TYPE _eDbmText : (txt_DbVar_C0_RamEcuInputsC0_PressureBlockOscillationState_0 := 0, txt_DbVar_C0_RamEcuInputsC0_PressureBlockOscillationValue_0 := 1, txt_DbVar_C0_RamEcuInputsC0_PressureBlockOscillationRawValue_0 := 2, txt_DbVar_C0_RamEcuInputsC0_PressureBrakeSensorState_0 := 3, txt_DbVar_C0_RamEcuInputsC0_PressureBrakeSensorValue_0 := 4, txt_DbVar_C0_RamEcuInputsC0_PressureBrakeSensorRawValue_0 := 5, txt_DbVar_C0_RamEcuInputsC0_TemperatureTransmissionState_0 := 6, txt_DbVar_C0_RamEcuInputsC0_TemperatureTransmissionValue_0 := 7, txt_DbVar_C0_RamEcuInputsC0_TemperatureTransmissionRawValue_0 := 8, txt_DbVar_C0_RamEcuInputsC0_FaultPvgLeftTrakState_0 := 9, txt_DbVar_C0_RamEcuInputsC0_FaultPvgLeftTrakRawValue_0 := 10, txt_DbVar_C0_RamEcuInputsC0_FaultPvgRightTrakState_0 := 11, txt_DbVar_C0_RamEcuInputsC0_FaultPvgRightTrakRawValue_0 := 12, txt_DbVar_C0_RamEcuInputsC0_DownAxleOscillantState_0 := 13, txt_DbVar_C0_RamEcuInputsC0_DownAxleOscillantRawValuePin0_0 := 14, txt_DbVar_C0_RamEcuInputsC0_DownAxleOscillantRawValuePin1_0 := 15, txt_DbVar_C0_RamEcuInputsC0_DownAxleFixeState_0 := 16, txt_DbVar_C0_RamEcuInputsC0_DownAxleFixeRawValuePin0_0 := 17, txt_DbVar_C0_RamEcuInputsC0_DownAxleFixeRawValuePin1_0 := 18, txt_DbVar_C0_RamEcuInputsC0_UpAxleOscillantState_0 := 19, txt_DbVar_C0_RamEcuInputsC0_UpAxleOscillantRawValue_0 := 20, txt_DbVar_C0_RamEcuInputsC0_UpAxleFixeState_0 := 21, txt_DbVar_C0_RamEcuInputsC0_UpAxleFixeRawValue_0 := 22, txt_DbVar_C0_RamEcuInputsC0_FrameRotationSensor1State_0 := 23, txt_DbVar_C0_RamEcuInputsC0_FrameRotationSensor1RawValuePin0_0 := 24, txt_DbVar_C0_RamEcuInputsC0_FrameRotationSensor1RawValuePin1_0 := 25, txt_DbVar_C0_RamEcuInputsC0_RailHookSensorState_0 := 26, txt_DbVar_C0_RamEcuInputsC0_RailHookSensorRawValue_0 := 27, txt_DbVar_C0_RamEcuInputsC0_InductiveRailSensorState_0 := 28, txt_DbVar_C0_RamEcuInputsC0_InductiveRailSensorRawValue_0 := 29, txt_DbVar_C0_RamEcuInputsC0_CenteredTurretState_0 := 30, txt_DbVar_C0_RamEcuInputsC0_CenteredTurretRawValue_0 := 31, txt_DbVar_C0_RamEcuInputsC0_WorkKeyTrackSideState_0 := 32, txt_DbVar_C0_RamEcuInputsC0_WorkKeyTrackSideRawValue_0 := 33, txt_DbVar_C0_RamEcuInputsC0_FrameRotationSensor2State_0 := 34, txt_DbVar_C0_RamEcuInputsC0_FrameRotationSensor2RawValuePin0_0 := 35, txt_DbVar_C0_RamEcuInputsC0_FrameRotationSensor2RawValuePin1_0 := 36, txt_DbVar_C0_RamEcuInputsC0_WorkKeyBilateralState_0 := 37, txt_DbVar_C0_RamEcuInputsC0_WorkKeyBilateralRawValue_0 := 38, txt_DbVar_C0_RamEcuInputsC0_WorkKeyCentredState_0 := 39, txt_DbVar_C0_RamEcuInputsC0_WorkKeyCentredRawValue_0 := 40, txt_DbVar_C0_RamEcuInputsC0_AbutmentTurretTrackSideState_0 := 41, txt_DbVar_C0_RamEcuInputsC0_AbutmentTurretTrackSideRaw_0 := 42, txt_DbVar_C0_RamEcuInputsC0_AbutmentTurretCentredSideState_0 := 43, txt_DbVar_C0_RamEcuInputsC0_AbutmentTurretCentredSideRaw_0 := 44, txt_DbVar_C0_RamEcuInputsC0_OscillantAxleSpeedSensorDirState_0 := 45, txt_DbVar_C0_RamEcuInputsC0_OscillantAxleSpeedSensorDirRaw_0 := 46, txt_DbVar_C0_RamEcuInputsC0_FixeAxleSpeedSensorDirState_0 := 47, txt_DbVar_C0_RamEcuInputsC0_FixeAxleSpeedSensorDirRaw_0 := 48, txt_DbVar_C0_RamEcuInputsC0_TrailerGacheState_0 := 49, txt_DbVar_C0_RamEcuInputsC0_TrailerGacheRawValue_0 := 50, txt_DbVar_C0_RamEcuInputsC0_MeasuringMastSensorFoldedState_0 := 51, txt_DbVar_C0_RamEcuInputsC0_MeasuringMastSensorFoldedRaw_0 := 52, txt_DbVar_C0_RamEcuInputsC0_OscillantAxleFrequency_0 := 53, txt_DbVar_C0_RamEcuInputsC0_FixeAxleFrequency_0 := 54, txt_DbVar_C0_RamEcuInputsC0_AruRadio1ContactState_0 := 55, txt_DbVar_C0_RamEcuInputsC0_AruRadio1ContactRawValue_0 := 56, txt_DbVar_C0_RamEcuInputsC0_AruRadio2ContactState_0 := 57, txt_DbVar_C0_RamEcuInputsC0_AruRadio2ContactRawValue_0 := 58, txt_DbVar_C0_RamEcuInputsC0_Aru1ContactState_0 := 59, txt_DbVar_C0_RamEcuInputsC0_Aru1ContactRawValue_0 := 60, txt_DbVar_C0_RamEcuInputsC0_Aru2ContactState_0 := 61, txt_DbVar_C0_RamEcuInputsC0_Aru2ContactRawValue_0 := 62, txt_DbVar_C0_RamEcuInputsC0_StarterMotorState_0 := 63, txt_DbVar_C0_RamEcuInputsC0_StarterMotorRawValue_0 := 64, txt_DbVar_C0_RamEcuInputsC0_AutorisationHighSpeedKeyState_0 := 65, txt_DbVar_C0_RamEcuInputsC0_AutorisationHighSpeedKeyRawValue_0 := 66, txt_DbVar_C0_RamEcuInputsC0_ElectricPumpPressureState_0 := 67, txt_DbVar_C0_RamEcuInputsC0_ElectricPumpPressureValue_0 := 68, txt_DbVar_C0_RamEcuInputsC0_ElectricPumpPressureRawValue_0 := 69, txt_DbVar_C0_RamEcuInputsC0_UpMastSensorNCState_0 := 70, txt_DbVar_C0_RamEcuInputsC0_UpMastSensorNCRawValue_0 := 71, txt_DbVar_C0_RamEcuInputsC0_ValveInDownPositionSensorState_0 := 72, txt_DbVar_C0_RamEcuInputsC0_ValveInDownPositionSensorValue_0 := 73, txt_DbVar_C0_RamEcuOutputsC0_EvDeflectorTransmissionCommand_0 := 74, txt_DbVar_C0_RamEcuOutputsC0_EvDeflectorTransmissionValue_0 := 75, txt_DbVar_C0_RamEcuOutputsC0_EvUpMeasuringMastCommand_0 := 76, txt_DbVar_C0_RamEcuOutputsC0_EvUpMeasuringMastValue_0 := 77, txt_DbVar_C0_RamEcuOutputsC0_EvDownMeasuringMastCommand_0 := 78, txt_DbVar_C0_RamEcuOutputsC0_EvDownMeasuringMastValue_0 := 79, txt_DbVar_C0_RamEcuOutputsC0_EvServiceBrakeTrackCommand_0 := 80, txt_DbVar_C0_RamEcuOutputsC0_EvServiceBrakeTrackValue_0 := 81, txt_DbVar_C0_RamEcuOutputsC0_EvPowerReductionCommand_0 := 82, txt_DbVar_C0_RamEcuOutputsC0_EvPowerReductionValue_0 := 83, txt_DbVar_C0_RamEcuOutputsC0_EvFrameRotation1Command_0 := 84, txt_DbVar_C0_RamEcuOutputsC0_EvFrameRotation1Value_0 := 85, txt_DbVar_C0_RamEcuOutputsC0_EvFrameRotation2Command_0 := 86, txt_DbVar_C0_RamEcuOutputsC0_EvFrameRotation2Value_0 := 87, txt_DbVar_C0_RamEcuOutputsC0_SupplyRadioReceiverCommand_0 := 88, txt_DbVar_C0_RamEcuOutputsC0_SupplyRadioReceiverValue_0 := 89, txt_DbVar_C0_RamEcuOutputsC0_BuzzerLynxMovingMachineCommand_0 := 90, txt_DbVar_C0_RamEcuOutputsC0_BuzzerLynxMovingMachineValue_0 := 91, txt_DbVar_C0_RamEcuOutputsC0_WhiteLightsTrailerCommand_0 := 92, txt_DbVar_C0_RamEcuOutputsC0_WhiteLightsTrailerValue_0 := 93, txt_DbVar_C0_RamEcuOutputsC0_RedLightsTrailerCommand_0 := 94, txt_DbVar_C0_RamEcuOutputsC0_RedLightsTrailerValue_0 := 95, txt_DbVar_C0_RamEcuOutputsC0_WhiteLightAVGCommand_0 := 96, txt_DbVar_C0_RamEcuOutputsC0_WhiteLightAVGValue_0 := 97, txt_DbVar_C0_RamEcuOutputsC0_WhiteLightAVDCommand_0 := 98, txt_DbVar_C0_RamEcuOutputsC0_WhiteLightAVDValue_0 := 99, txt_DbVar_C0_RamEcuOutputsC0_RedLightAVGCommand_0 := 100, txt_DbVar_C0_RamEcuOutputsC0_RedLightAVGValue_0 := 101, txt_DbVar_C0_RamEcuOutputsC0_RedLightAVDCommand_0 := 102, txt_DbVar_C0_RamEcuOutputsC0_RedLightAVDValue_0 := 103, txt_DbVar_C0_RamEcuOutputsC0_WhiteLightARGCommand_0 := 104, txt_DbVar_C0_RamEcuOutputsC0_WhiteLightARGValue_0 := 105, txt_DbVar_C0_RamEcuOutputsC0_WhiteLightARDCommand_0 := 106, txt_DbVar_C0_RamEcuOutputsC0_WhiteLightARDValue_0 := 107, txt_DbVar_C0_RamEcuOutputsC0_RedLightARGCommand_0 := 108, txt_DbVar_C0_RamEcuOutputsC0_RedLightARGValue_0 := 109, txt_DbVar_C0_RamEcuOutputsC0_RedLightARDCommand_0 := 110, txt_DbVar_C0_RamEcuOutputsC0_RedLightARDValue_0 := 111, txt_DbVar_C0_RamEcuOutputsC0_SupllyPvgLeftTrackCommand_0 := 112, txt_DbVar_C0_RamEcuOutputsC0_SupllyPvgLeftTrackValue_0 := 113, txt_DbVar_C0_RamEcuOutputsC0_SupllyPvgRightTrackCommand_0 := 114, txt_DbVar_C0_RamEcuOutputsC0_SupllyPvgRightTrackValue_0 := 115, txt_DbVar_C0_RamEcuOutputsC0_EvUnBlockOscillationAxleState_0 := 116, txt_DbVar_C0_RamEcuOutputsC0_EvUnBlockOscillationAxleCmdBool_0 := 117, txt_DbVar_C0_RamEcuOutputsC0_EvUpAxleOscillantState_0 := 118, txt_DbVar_C0_RamEcuOutputsC0_EvUpAxleOscillantCommandBool_0 := 119, txt_DbVar_C0_RamEcuOutputsC0_EvDownAxleOscillantState_0 := 120, txt_DbVar_C0_RamEcuOutputsC0_EvDownAxleOscillantCommandBool_0 := 121, txt_DbVar_C0_RamEcuOutputsC0_EvUpAxleFixeState_0 := 122, txt_DbVar_C0_RamEcuOutputsC0_EvUpAxleFixeCommandBool_0 := 123, txt_DbVar_C0_RamEcuOutputsC0_EvDownAxleFixeState_0 := 124, txt_DbVar_C0_RamEcuOutputsC0_EvDownAxleFixeCommandBool_0 := 125, txt_DbVar_C0_RamEcuOutputsC0_EvParkBrakeAxleOscillantState_0 := 126, txt_DbVar_C0_RamEcuOutputsC0_EvParkBrakeAxleOscillantCmdBool_0 := 127, txt_DbVar_C0_RamEcuOutputsC0_EvParkBrakeAxleFixeState_0 := 128, txt_DbVar_C0_RamEcuOutputsC0_EvParkBrakeAxleFixeCmdBool_0 := 129, txt_DbVar_C0_RamEcuOutputsC0_EvServiceBrakeAxleOscillantState_0 := 130, txt_DbVar_C0_RamEcuOutputsC0_EvServiceBrakeAxleOsciCmdBool_0 := 131, txt_DbVar_C0_RamEcuOutputsC0_EvServiceBrakeAxleFixeState_0 := 132, txt_DbVar_C0_RamEcuOutputsC0_EvServiceBrakeAxleFixeCmdBool_0 := 133, txt_DbVar_C0_RamEcuOutputsC0_KlaxonNeotecState_0 := 134, txt_DbVar_C0_RamEcuOutputsC0_KlaxonNeotecCmdBool_0 := 135, txt_DbVar_C0_RamEcuOutputsC0_ForwardPumpState_0 := 136, txt_DbVar_C0_RamEcuOutputsC0_ForwardPumpCommand_0 := 137, txt_DbVar_C0_RamEcuOutputsC0_ForwardPumpCurrent_0 := 138, txt_DbVar_C0_RamEcuOutputsC0_BackwardPumpState_0 := 139, txt_DbVar_C0_RamEcuOutputsC0_BackwardPumpCommand_0 := 140, txt_DbVar_C0_RamEcuOutputsC0_BackwardPumpCurrent_0 := 141, txt_DbVar_C0_RamEcuOutputsC0_PvgLeftTrackCommand_0 := 142, txt_DbVar_C0_RamEcuOutputsC0_PvgLeftTrackVoltage_0 := 143, txt_DbVar_C0_RamEcuOutputsC0_PvgRightTrackCommand_0 := 144, txt_DbVar_C0_RamEcuOutputsC0_PvgRightTrackVoltage_0 := 145, txt_DbVar_C0_RamEcuOutputsC0_SupplyAnaSensorsCommand_0 := 146, txt_DbVar_C0_RamEcuOutputsC0_SupplyAnaSensorsValue_0 := 147, txt_DbVar_C0_RamEcuOutputsC0_PvgLeftTrackLowsideCommand_0 := 148, txt_DbVar_C0_RamEcuOutputsC0_PvgLeftTrackLowsideValue_0 := 149, txt_DbVar_C0_RamEcuOutputsC0_PvgRightTrackLowsideCommand_0 := 150, txt_DbVar_C0_RamEcuOutputsC0_PvgRightTrackLowsideValue_0 := 151, txt_DbVar_C0_RamEcuOutputsC0_ReturnLowSideEvForwardPumpCmd_0 := 152, txt_DbVar_C0_RamEcuOutputsC0_ReturnLowSideEvForwardPumpState_0 := 153, txt_DbVar_C0_RamEcuOutputsC0_ReturnLowSideEvBackwardPumpCmd_0 := 154, txt_DbVar_C0_RamEcuOutputsC0_ReturnLowSideEvBackwardPumpState_0 := 155, txt_DbVar_C0_RamEcuOutputsC0_NeonLightsCmd_0 := 156, txt_DbVar_C0_RamEcuOutputsC0_NeonLightsValue_0 := 157, txt_DbVar_C0_RamEcuOutputsC0_Ev2DeflectorTransmissionValue_0 := 158, txt_DbVar_C0_RamEcuOutputsC0_CoolingRelayCommand_0 := 159, txt_DbVar_C0_RamEcuOutputsC0_CoolingRelayState_0 := 160, txt_DbVar_C0_RamEcuOutputsC0_Ev2ndParkBrakeAxleFixe_0 := 161, txt_DbVar_C0_RamEcuOutputsC0_Ev2ndParkBrakeAxleOsci_0 := 162, txt_DbVar_C0_RamEcuOutputsC0_Ev2ndParkBrakeAxleFixeState_0 := 163, txt_DbVar_C0_RamEcuOutputsC0_Ev2ndParkBrakeAxleOsciState_0 := 164, txt_DbVar_C0_RamEcuOutputsC0_PvgTransRailElectricCmd_0 := 165, txt_DbVar_C0_RamEcuOutputsC0_PvgTransRailElectricVoltage_0 := 166, txt_DbVar_C0_RamEcuOutputsC0_SupllyPvgTransRailElectricCmd_0 := 167, txt_DbVar_C0_RamEcuOutputsC0_SupllyPvgTransRailElectricState_0 := 168, txt_DbVar_C0_RamEcuOutputsC0_EvDevRailElectricModeCmd_0 := 169, txt_DbVar_C0_RamEcuOutputsC0_EvDevRailElectricModeState_0 := 170, txt_DbVar_C0_RamEcuOutputsC0_RelayCutOffVariatorElectricCmd_0 := 171, txt_DbVar_C0_RamEcuOutputsC0_RelayCutOffVariatorElectricState_0 := 172, txt_DbVar_C0_RamEcuOutputsC0_RelayEnableBatteryCmd_0 := 173, txt_DbVar_C0_RamEcuOutputsC0_RelayEnableBatteryState_0 := 174, txt_DbVar_C0_RamGeneralC0_LifeByte_0 := 175, txt_DbVar_C0_RamGeneralC0_WatchdogState_0 := 176, txt_DbVar_C0_RamGeneralC0_EcuVoltage_0 := 177, txt_DbVar_C0_RamGeneralC0_OffRailMode_0 := 178, txt_DbVar_C0_RamGeneralC0_RailSpeedMode_0 := 179, txt_DbVar_C0_RamGeneralC0_OutputLutLeftManipulator_0 := 180, txt_DbVar_C0_RamGeneralC0_OutputLutLeftTrackPvg_0 := 181, txt_DbVar_C0_RamGeneralC0_OutputLutRightManipulator_0 := 182, txt_DbVar_C0_RamGeneralC0_OutputLutRightTrackPvg_0 := 183, txt_DbVar_C0_RamGeneralC0_OutputLutJoystickAdvanceRail_0 := 184, txt_DbVar_C0_RamGeneralC0_OutputLutForwardPumpTransmission_0 := 185, txt_DbVar_C0_RamGeneralC0_OutputLutBackwardPumpTransm_0 := 186, txt_DbVar_C0_RamGeneralC0_ConsigneForwardPumpTransmPercent_0 := 187, txt_DbVar_C0_RamGeneralC0_LastJoystickAdvanceValue_0 := 188, txt_DbVar_C0_RamGeneralC0_JoystickAdvanceScalingValue_0 := 189, txt_DbVar_C0_RamGeneralC0_StateServiceBrakeRail_0 := 190, txt_DbVar_C0_RamGeneralC0_EnableStartTimerServiceBrake_0 := 191, txt_DbVar_C0_RamGeneralC0_SpeedMotorCommandTest_0 := 192, txt_DbVar_C0_RamGeneralC0_ForceSilentModeMotorTest_0 := 193, txt_DbVar_C0_RamGeneralC0_AngularSensorTest_0 := 194, txt_DbVar_C0_RamGeneralC0_SpeedAxleSensor_0 := 195, txt_DbVar_C0_RamGeneralC0_AverageTimeCycle_0 := 196, txt_DbVar_C0_RamGeneralC0_MaxTimeCycle_0 := 197, txt_DbVar_C0_RamGeneralC0_FirstTranslationReleaseParkBrake_0 := 198, txt_DbVar_C0_RamGeneralC0_AutorizeUpAxleOscillant_0 := 199, txt_DbVar_C0_RamGeneralC0_AutorizeDownAxleOscillant_0 := 200, txt_DbVar_C0_RamGeneralC0_AutorizeUpAxlefixe_0 := 201, txt_DbVar_C0_RamGeneralC0_AutorizeDownAxlefixe_0 := 202, txt_DbVar_C0_RamGeneralC0_EngineOn_0 := 203, txt_DbVar_C0_RamGeneralC0_TranslationMovementIsSolicited_0 := 204, txt_DbVar_C0_RamGeneralC0_RailTranslationDirection_0 := 205, txt_DbVar_C0_RamGeneralC0_SetConditionAruRadioAlarm_0 := 206, txt_DbVar_C0_RamGeneralC0_JoystickAdvanceSetpointAfterRamp_0 := 207, txt_DbVar_C0_RamGeneralC0_StabilizedStop_0 := 208, txt_DbVar_C0_RamGeneralC0_EmergencyBrake_0 := 209, txt_DbVar_C0_RamGeneralC0_EmergencyServiceBrakeTimerDone_0 := 210, txt_DbVar_C0_RamGeneralC0_StoppedMachineUnblkOsciTimerDone_0 := 211, txt_DbVar_C0_RamGeneralC0_OutLutLeftManipulatorAfterRamp_0 := 212, txt_DbVar_C0_RamGeneralC0_OutLutRightManipulatorAfterRamp_0 := 213, txt_DbVar_C0_RamGeneralC0_DeltaBeetweenLeftRightPvgCrawler_0 := 214, txt_DbVar_C0_RamGeneralC0_ConsigneLeftPvgTrack_0 := 215, txt_DbVar_C0_RamGeneralC0_ConsigneRightPvgTrack_0 := 216, txt_DbVar_C0_RamGeneralC0_BrakeWithoutGachetteOrPedal_0 := 217, txt_DbVar_C0_RamGeneralC0_AruRadioAlarmCounter_0 := 218, txt_DbVar_C0_RamGeneralC0_RedLightARGBasketCmd_0 := 219, txt_DbVar_C0_RamGeneralC0_WhiteLightARGBasketCmd_0 := 220, txt_DbVar_C0_RamGeneralC0_PortillonLadderClose_0 := 221, txt_DbVar_C0_RamGeneralC0_TestEvision_0 := 222, txt_DbVar_C0_RamGeneralC0_PosJoystickAdvance_0 := 223, txt_DbVar_C0_RamGeneralC0_RetainPosJoyAdvanceUntilBrake_0 := 224, txt_DbVar_C0_RamGeneralC0_AuthorizeForwardCrawler_0 := 225, txt_DbVar_C0_RamGeneralC0_AuthorizeBackwardCrawler_0 := 226, txt_DbVar_C0_RamGeneralC0_ReturnValueUartInit_0 := 227, txt_DbVar_C0_RamGeneralC0_AuthorizeTransRailMovement_0 := 228, txt_DbVar_C0_RamGeneralC0_EvForwardTrackConsigne_0 := 229, txt_DbVar_C0_RamGeneralC0_EvForwardRailConsigne_0 := 230, txt_DbVar_C0_RamGeneralC0_EngineTimeSecond_0 := 231, txt_DbVar_C0_RamGeneralC0_RamGeneralNeotecC0_1_0 := 232, txt_DbVar_C0_RamGeneralC0_RamGeneralNeotecC0_1_1_0 := 233, txt_DbVar_C0_RamGeneralC0_RamGeneralNeotecC0_1_2_0 := 234, txt_DbVar_C0_RamGeneralC0_RamGeneralNeotecC0_1_3_0 := 235, txt_DbVar_C0_RamGeneralC0_RamGeneralNeotecC0_1_4_0 := 236, txt_DbVar_C0_RamGeneralC0_RamGeneralNeotecC0_1_5_0 := 237, txt_DbVar_C0_RamGeneralC0_RamGeneralNeotecC0_1_6_0 := 238, txt_DbVar_C0_RamGeneralC0_RamGeneralNeotecC0_1_7_0 := 239, txt_DbVar_C0_RamGeneralC0_RamGeneralNeotecC0_1_8_0 := 240, txt_DbVar_C0_RamGeneralC0_RamGeneralNeotecC0_1_9_0 := 241, txt_DbVar_C0_RamGeneralC0_RamGeneralNeotecC0_1_10_0 := 242, txt_DbVar_C0_RamGeneralC0_RamGeneralNeotecC0_1_11_0 := 243, txt_DbVar_C0_RamGeneralC0_RamGeneralNeotecC0_1_12_0 := 244, txt_DbVar_C0_RamGeneralC0_RamGeneralNeotecC0_1_13_0 := 245, txt_DbVar_C0_RamGeneralC0_RamGeneralNeotecC0_1_14_0 := 246, txt_DbVar_C0_RamGeneralC0_RamGeneralNeotecC0_1_15_0 := 247, txt_DbVar_C0_RamGeneralC0_RamGeneralNeotecC0_2_0 := 248, txt_DbVar_C0_RamGeneralC0_RamGeneralNeotecC0_2_1_0 := 249, txt_DbVar_C0_RamGeneralC0_RamGeneralNeotecC0_2_2_0 := 250, txt_DbVar_C0_RamGeneralC0_RamGeneralNeotecC0_2_3_0 := 251, txt_DbVar_C0_RamGeneralC0_RamGeneralNeotecC0_2_4_0 := 252, txt_DbVar_C0_RamGeneralC0_RamGeneralNeotecC0_2_5_0 := 253, txt_DbVar_C0_RamGeneralC0_RamGeneralNeotecC0_3_0 := 254, txt_DbVar_C0_RamGeneralC0_RamGeneralNeotecC0_3_1_0 := 255, txt_DbVar_C0_RamGeneralC0_RamGeneralNeotecC0_3_2_0 := 256, txt_DbVar_C0_RamGeneralC0_RamGeneralNeotecC0_3_3_0 := 257, txt_DbVar_C0_RamGeneralC0_RamGeneralNeotecC0_3_4_0 := 258, txt_DbVar_C0_RamGeneralC0_RamGeneralNeotecC0_3_5_0 := 259, txt_DbVar_C0_RamGeneralC0_RamGeneralNeotecC0_3_6_0 := 260, txt_DbVar_C0_RamGeneralC0_RamGeneralNeotecC0_3_7_0 := 261, txt_DbVar_C0_RamGeneralC0_RamGeneralNeotecC0_3_8_0 := 262, txt_DbVar_C0_RamGeneralC0_RamGeneralNeotecC0_4_0 := 263, txt_DbVar_C0_RamGeneralC0_RamGeneralNeotecC0_4_1_0 := 264, txt_DbVar_C0_RamGeneralC0_RamGeneralNeotecC0_4_2_0 := 265, txt_DbVar_C0_RamGeneralC0_RamGeneralNeotecC0_4_3_0 := 266, txt_DbVar_C0_RamGeneralC0_RamGeneralNeotecC0_4_4_0 := 267, txt_DbVar_C0_RamGeneralC0_RamGeneralNeotecC0_4_5_0 := 268, txt_DbVar_C0_RamGeneralC0_RamGeneralNeotecC0_4_6_0 := 269, txt_DbVar_C0_RamGeneralC0_RamGeneralNeotecC0_4_7_0 := 270, txt_DbVar_C0_RamGeneralC0_RamGeneralNeotecC0_4_8_0 := 271, txt_DbVar_C0_RamGeneralC0_RedLightARDBasketCmd_0 := 272, txt_DbVar_C0_RamGeneralC0_WhiteLightARDBasketCmd_0 := 273, txt_DbVar_C0_RamGeneralC0_ActiveFailure_0 := 274, txt_DbVar_C0_RamGeneralC0_ReductionPumpRail_0 := 275, txt_DbVar_C0_RamGeneralC0_ReductionPumpTrack_0 := 276, txt_DbVar_C0_RamGeneralC0_ActiveWhiteLights15746_0 := 277, txt_DbVar_C0_RamGeneralC0_WhiteLightAv15746Command_0 := 278, txt_DbVar_C0_RamGeneralC0_WhiteLightAr15746Command_0 := 279, txt_DbVar_C0_RamGeneralC0_TestElectricalIO_0 := 280, txt_DbVar_C0_RamGeneralC0_SendEventDataloggerMessage_0 := 281, txt_DbVar_C0_RamGeneralC0_SlopeModeFromC1_0 := 282, txt_DbVar_C0_RamGeneralC0_BlinkLow_0 := 283, txt_DbVar_C0_RamGeneralC0_TotalDistance_0 := 284, txt_DbVar_C0_RamGeneralC0_RunningStable48XS_0 := 285, txt_DbVar_C0_RamGeneralC0_AlarmHydTempRailActive_0 := 286, txt_DbVar_C0_RamGeneralC0_AlarmHydTempCrawlerActive_0 := 287, txt_DbVar_C0_RamGeneralC0_FaultyValue_0 := 288, txt_DbVar_C0_RamGeneralC0_DeviceNum_0 := 289, txt_DbVar_C0_RamGeneralC0_ErrorCode_0 := 290, txt_DbVar_C0_RamGeneralC0_EngineRunningStable_0 := 291, txt_DbVar_C0_NvOptionsC0_ConfigHollandaise_0 := 292, txt_DbVar_C0_NvOptionsC0_Portillon_0 := 293, txt_DbVar_C0_NvOptionsC0_Ladder_0 := 294, txt_DbVar_C0_NvOptionsC0_MeasuringMat_0 := 295, txt_DbVar_C0_NvOptionsC0_IncliBasketHighSectorForAcesSite_0 := 296, txt_DbVar_C0_NvOptionsC0_BasketCenteredForAccesSite_0 := 297, txt_DbVar_C0_NvOptionsC0_MastDigitalDisplay_0 := 298, txt_DbVar_C0_NvOptionsC0_AutorisationWorkKeyPresent_0 := 299, txt_DbVar_C0_NvOptionsC0_SecondParkBrakeActive_0 := 300, txt_DbVar_C0_NvOptionsC0_AddPerformanceFunc_0 := 301, txt_DbVar_C0_NvOptionsC0_BasketTurretLimitation_0 := 302, txt_DbVar_C0_NvOptionsC0_PresenceSensorPlate_0 := 303, txt_DbVar_C0_NvMemoryC0_NCycleBrakePerform_0 := 304, txt_DbVar_C0_NvMemoryC0_LightMode_0 := 305, txt_DbVar_C0_NvMemoryC0_VarMemory1_0 := 306, txt_DbVar_C0_NvMemoryC0_VarMemory2_0 := 307, txt_DbVar_C0_NvMemoryC0_VarMemory3_0 := 308, txt_DbVar_C0_NvMemoryC0_VarMemory4_0 := 309, txt_DbVar_C0_NvMemoryC0_VarMemory5_0 := 310, txt_DbVar_C0_NvMemoryC0_VarMemory6_0 := 311, txt_DbVar_C0_NvMemoryC0_VarMemory7_0 := 312, txt_DbVar_C0_NvMemoryC0_VarMemory8_0 := 313, txt_DbVar_C0_NvMemoryC0_VarMemory9_0 := 314, txt_DbVar_C0_NvMemoryC0_VarMemory10_0 := 315, txt_DbVar_C0_NvMemoryC0_VarMemory11_0 := 316, txt_DbVar_C0_NvMemoryC0_VarMemory12_0 := 317, txt_DbVar_C0_NvMemoryC0_VarMemory13_0 := 318, txt_DbVar_C0_NvMemoryC0_VarMemory14_0 := 319, txt_DbVar_C0_NvMemoryC0_gDistanceTraveledMeasureMast_0 := 320, txt_DbVar_C0_NvMemoryC0_NCycle2ndParkBrakePerform_0 := 321, txt_DbVar_C0_NvMemoryC0_gTotalDistanceMsb_0 := 322, txt_DbVar_C0_NvMemoryC0_gTotalDistanceLsb_0 := 323, txt_DbVar_C0_NvParametersC0_LimitTresholdAngleRadioControl_0 := 324, txt_DbVar_C0_NvParametersC0_TresholdMinimalSpeedParkBrake_0 := 325, txt_DbVar_C0_NvParametersC0_TresholdMinimalSpeedServiceBrake_0 := 326, txt_DbVar_C0_NvParametersC0_AdditionnalPourcentFwardPumpCmd_0 := 327, txt_DbVar_C0_NvParametersC0_AddPrctFwardPumpSilentModeMotor_0 := 328, txt_DbVar_C0_NvParametersC0_NodeIdRadioCommand_0 := 329, txt_DbVar_C0_NvParametersC0_DeadZoneJoystickRotationTurret_0 := 330, txt_DbVar_C0_NvParametersC0_ServiceAxleBrakeTimeBeforeBrake_0 := 331, txt_DbVar_C0_NvParametersC0_ServiceBrakeOffrailTime_0 := 332, txt_DbVar_C0_NvParametersC0_EngineOffCurEvForwardPump_0 := 333, txt_DbVar_C0_NvParametersC0_MinCurEvForwardPump_0 := 334, txt_DbVar_C0_NvParametersC0_StopCurEvForwardPump_0 := 335, txt_DbVar_C0_NvParametersC0_EngineOffCurEvBackwardPump_0 := 336, txt_DbVar_C0_NvParametersC0_MinCurEvBackwardPump_0 := 337, txt_DbVar_C0_NvParametersC0_StopCurEvBackwardPump_0 := 338, txt_DbVar_C0_NvParametersC0_PosNeutralJoyAdvancement_0 := 339, txt_DbVar_C0_NvParametersC0_PidGpEvForwardPump_0 := 340, txt_DbVar_C0_NvParametersC0_PidTiEvForwardPump_0 := 341, txt_DbVar_C0_NvParametersC0_PidTdEvForwardPump_0 := 342, txt_DbVar_C0_NvParametersC0_PidGpEvBackwardPump_0 := 343, txt_DbVar_C0_NvParametersC0_PidTiEvBackwardPump_0 := 344, txt_DbVar_C0_NvParametersC0_PidTdEvBackwardPump_0 := 345, txt_DbVar_C0_NvParametersC0_OutCharPosPressureBlockOscil_0 := 346, txt_DbVar_C0_NvParametersC0_OutCharNeuPressureBlockOscil_0 := 347, txt_DbVar_C0_NvParametersC0_OutCharNegPressureBlockOscil_0 := 348, txt_DbVar_C0_NvParametersC0_OutCharPosPressureBrake_0 := 349, txt_DbVar_C0_NvParametersC0_OutCharNeuPressureBrake_0 := 350, txt_DbVar_C0_NvParametersC0_OutCharNegPressureBrake_0 := 351, txt_DbVar_C0_NvParametersC0_OutCharPosTempTransmission_0 := 352, txt_DbVar_C0_NvParametersC0_OutCharNeuTempTransmission_0 := 353, txt_DbVar_C0_NvParametersC0_OutCharNegTempTransmission_0 := 354, txt_DbVar_C0_NvParametersC0_MinConsigneEvForwardRail_0 := 355, txt_DbVar_C0_NvParametersC0_MaxConsigneEvForwardRail_0 := 356, txt_DbVar_C0_NvParametersC0_MinConsigneEvBackwardRail_0 := 357, txt_DbVar_C0_NvParametersC0_MaxConsigneEvBackwardRail_0 := 358, txt_DbVarArrDescr_C0_NvParametersC0_TimeRampEvAdvancementRail := 359, txt_DbVar_C0_NvParametersC0_TimeRampEvAdvancementRail_0 := 360, txt_DbVar_C0_NvParametersC0_TimeRampEvAdvancementRail_1 := 361, txt_DbVar_C0_NvParametersC0_TimeRampEvAdvancementRail_2 := 362, txt_DbVar_C0_NvParametersC0_TimeRampEvAdvancementRail_3 := 363, txt_DbVar_C0_NvParametersC0_MinConsigneEvForwardCrawler_0 := 364, txt_DbVar_C0_NvParametersC0_MaxConsigneEvForwardCrawler_0 := 365, txt_DbVarArrDescr_C0_NvParametersC0_EvForwardCrawlerAdvanceRampRatio := 366, txt_DbVar_C0_NvParametersC0_EvForwardCrawlerAdvanceRampRatio_0 := 367, txt_DbVar_C0_NvParametersC0_EvForwardCrawlerAdvanceRampRatio_1 := 368, txt_DbVar_C0_NvParametersC0_TresholdRegimeMotorParkBrake_0 := 369, txt_DbVar_C0_NvParametersC0_MinPvgLeftTrackAv_0 := 370, txt_DbVar_C0_NvParametersC0_MaxPvgLeftTrackAv_0 := 371, txt_DbVar_C0_NvParametersC0_MinPvgLeftTrackAr_0 := 372, txt_DbVar_C0_NvParametersC0_MaxPvgLeftTrackAr_0 := 373, txt_DbVar_C0_NvParametersC0_MinPvgRightTrackAv_0 := 374, txt_DbVar_C0_NvParametersC0_MaxPvgRightTrackAv_0 := 375, txt_DbVar_C0_NvParametersC0_MinPvgRightTrackAr_0 := 376, txt_DbVar_C0_NvParametersC0_MaxPvgRightTrackAr_0 := 377, txt_DbVarArrDescr_C0_NvParametersC0_TimeRampLeftTrack := 378, txt_DbVar_C0_NvParametersC0_TimeRampLeftTrack_0 := 379, txt_DbVar_C0_NvParametersC0_TimeRampLeftTrack_1 := 380, txt_DbVar_C0_NvParametersC0_TimeRampLeftTrack_2 := 381, txt_DbVar_C0_NvParametersC0_TimeRampLeftTrack_3 := 382, txt_DbVarArrDescr_C0_NvParametersC0_TimeRampRightTrack := 383, txt_DbVar_C0_NvParametersC0_TimeRampRightTrack_0 := 384, txt_DbVar_C0_NvParametersC0_TimeRampRightTrack_1 := 385, txt_DbVar_C0_NvParametersC0_TimeRampRightTrack_2 := 386, txt_DbVar_C0_NvParametersC0_TimeRampRightTrack_3 := 387, txt_DbVar_C0_NvParametersC0_TimeStabilizedStopDetection_0 := 388, txt_DbVar_C0_NvParametersC0_TresholdLowSpeedStabilizedStop_0 := 389, txt_DbVar_C0_NvParametersC0_TimeEmergencyServiceBrake_0 := 390, txt_DbVar_C0_NvParametersC0_TimeStoppedMachineUnblockOscAxle_0 := 391, txt_DbVar_C0_NvParametersC0_TresholdLowSpeedUnblockOsciAxle_0 := 392, txt_DbVar_C0_NvParametersC0_GapMaxPvgCrawlerAdvancement_0 := 393, txt_DbVar_C0_NvParametersC0_GapMaxInvertedPvgCrawler_0 := 394, txt_DbVar_C0_NvParametersC0_TresholdAnaToBoForInputs48Xs_0 := 395, txt_DbVar_C0_NvParametersC0_InMinJoystickAdvance_0 := 396, txt_DbVar_C0_NvParametersC0_InMaxJoystickAdvance_0 := 397, txt_DbVar_C0_NvParametersC0_SpeedMiniTresholdServiceBrake_0 := 398, txt_DbVar_C0_NvParametersC0_NbElementAverageSlopeTransAngle_0 := 399, txt_DbVar_C0_NvParametersC0_NbElementAverageSlopeLongAngle_0 := 400, txt_DbVar_C0_NvParametersC0_DeadZoneJoystickRailAdvancement_0 := 401, txt_DbVar_C0_NvParametersC0_NbElementAverageSlopeTransAngle2_0 := 402, txt_DbVar_C0_NvParametersC0_NbElementAverageSlopeLongAngle2_0 := 403, txt_DbVar_C0_NvParametersC0_NvParametersC0_1_0 := 404, txt_DbVar_C0_NvParametersC0_NvParametersC0_2_0 := 405, txt_DbVar_C0_NvParametersC0_NvParametersC0_3_0 := 406, txt_DbVar_C0_NvParametersC0_NvParametersC0_4_0 := 407, txt_DbVar_C0_NvParametersC0_NvParametersC0_5_0 := 408, txt_DbVar_C0_NvParametersC0_NvParametersC0_6_0 := 409, txt_DbVar_C0_NvParametersC0_NvParametersC0_7_0 := 410, txt_DbVar_C0_NvParametersC0_NvParametersC0_8_0 := 411, txt_DbVar_C0_NvParametersC0_NvParametersC0_9_0 := 412, txt_DbVar_C0_NvParametersC0_NvParametersC0_10_0 := 413, txt_DbVar_C0_NvParametersC0_NvParametersC0_11_0 := 414, txt_DbVar_C0_NvParametersC0_NvParametersC0_12_0 := 415, txt_DbVar_C0_NvParametersC0_NvParametersC0_13_0 := 416, txt_DbVar_C0_NvParametersC0_NvParametersC0_14_0 := 417, txt_DbVar_C0_NvParametersC0_NvParametersC0_15_0 := 418, txt_DbVar_C0_NvParametersC0_NvParametersC0_16_0 := 419, txt_DbVar_C0_NvParametersC0_NvParametersC0_17_0 := 420, txt_DbVar_C0_NvParametersC0_ThreshotothydraulicTemperature_0 := 421, txt_DbVar_C0_NvParametersC0_TimeforCoolerOn_0 := 422, txt_DbVar_C0_NvParametersC0_TimeFaultPressureReducCrawler_0 := 423, txt_DbVar_C0_NvParametersC0_RailJoyRatioTwoSpeedFault_0 := 424, txt_DbVar_C0_NvParametersC0_TimeoutSdoRequestTime_0 := 425, txt_DbVar_C0_NvParametersC0_PeriodBlinkoffWhiteLight_0 := 426, txt_DbVar_C0_NvParametersC0_CptNeutralJoystickMax_0 := 427, txt_DbVar_C0_NvParametersC0_StopMotorMGmax_0 := 428, txt_DbVar_C0_NvParametersC0_TurretRearPosExtLowSpeedTresh_0 := 429, txt_DbVar_C0_NvParametersC0_TurretRearNegExtLowSpeedTresh_0 := 430, txt_DbVar_C0_NvParametersC0_NbOfFileParameters_0 := 431, txt_DbVar_C0_NvParametersC0_VersionMajor_0 := 432, txt_DbVar_C0_NvParametersC0_VersionMinior_0 := 433, txt_DbVar_C0_NvParametersC0_VersionPatch_0 := 434, txt_DbVar_C0_NvParametersC0_VersionCustom_0 := 435, txt_DbVar_C0_NvParametersC0_OutCharPosElectricPumpPressure_0 := 436, txt_DbVar_C0_NvParametersC0_OutCharNeuElectricPumpPressure_0 := 437, txt_DbVar_C0_NvParametersC0_OutCharNegElectricPumpPressure_0 := 438, txt_DbVar_C0_NvCalibrationC0_ManipulatorLeftMaxPointLut_0 := 439, txt_DbVarArrDescr_C0_NvCalibrationC0_ManipulatorLeftXValue := 440, txt_DbVar_C0_NvCalibrationC0_ManipulatorLeftXValue_0 := 441, txt_DbVar_C0_NvCalibrationC0_ManipulatorLeftXValue_1 := 442, txt_DbVarArrDescr_C0_NvCalibrationC0_ManipulatorLeftYValue := 443, txt_DbVar_C0_NvCalibrationC0_ManipulatorLeftYValue_0 := 444, txt_DbVar_C0_NvCalibrationC0_ManipulatorLeftYValue_1 := 445, txt_DbVar_C0_NvCalibrationC0_ManipulatorRightMaxPointLut_0 := 446, txt_DbVarArrDescr_C0_NvCalibrationC0_ManipulatorRightXValue := 447, txt_DbVar_C0_NvCalibrationC0_ManipulatorRightXValue_0 := 448, txt_DbVar_C0_NvCalibrationC0_ManipulatorRightXValue_1 := 449, txt_DbVarArrDescr_C0_NvCalibrationC0_ManipulatorRightYValue := 450, txt_DbVar_C0_NvCalibrationC0_ManipulatorRightYValue_0 := 451, txt_DbVar_C0_NvCalibrationC0_ManipulatorRightYValue_1 := 452, txt_DbVar_C0_NvCalibrationC0_LeftTrackPvgMaxPointLut_0 := 453, txt_DbVarArrDescr_C0_NvCalibrationC0_LeftTrackPvgRampRatio := 454, txt_DbVar_C0_NvCalibrationC0_LeftTrackPvgRampRatio_0 := 455, txt_DbVar_C0_NvCalibrationC0_LeftTrackPvgRampRatio_1 := 456, txt_DbVarArrDescr_C0_NvCalibrationC0_RangeValueOfLeftTrackPvgRamp := 457, txt_DbVar_C0_NvCalibrationC0_RangeValueOfLeftTrackPvgRamp_0 := 458, txt_DbVar_C0_NvCalibrationC0_RangeValueOfLeftTrackPvgRamp_1 := 459, txt_DbVar_C0_NvCalibrationC0_RangeValueOfLeftTrackPvgRamp_2 := 460, txt_DbVarArrDescr_C0_NvCalibrationC0_RightTrackPvgRampRatio := 461, txt_DbVar_C0_NvCalibrationC0_RightTrackPvgRampRatio_0 := 462, txt_DbVar_C0_NvCalibrationC0_RightTrackPvgRampRatio_1 := 463, txt_DbVarArrDescr_C0_NvCalibrationC0_RangeValueOfRightTrackPvgRamp := 464, txt_DbVar_C0_NvCalibrationC0_RangeValueOfRightTrackPvgRamp_0 := 465, txt_DbVar_C0_NvCalibrationC0_RangeValueOfRightTrackPvgRamp_1 := 466, txt_DbVar_C0_NvCalibrationC0_RangeValueOfRightTrackPvgRamp_2 := 467, txt_DbVar_C0_NvCalibrationC0_ForwardPumpTransmisMaxPointLut_0 := 468, txt_DbVarArrDescr_C0_NvCalibrationC0_ForwardPumpTransmissionXValue := 469, txt_DbVar_C0_NvCalibrationC0_ForwardPumpTransmissionXValue_0 := 470, txt_DbVar_C0_NvCalibrationC0_ForwardPumpTransmissionXValue_1 := 471, txt_DbVarArrDescr_C0_NvCalibrationC0_ForwardPumpTransmissionYValue := 472, txt_DbVar_C0_NvCalibrationC0_ForwardPumpTransmissionYValue_0 := 473, txt_DbVar_C0_NvCalibrationC0_ForwardPumpTransmissionYValue_1 := 474, txt_DbVar_C0_NvCalibrationC0_BackwardPumpTransmisMaxPointLut_0 := 475, txt_DbVarArrDescr_C0_NvCalibrationC0_BackwardPumpTransmissionXValue := 476, txt_DbVar_C0_NvCalibrationC0_BackwardPumpTransmissionXValue_0 := 477, txt_DbVar_C0_NvCalibrationC0_BackwardPumpTransmissionXValue_1 := 478, txt_DbVarArrDescr_C0_NvCalibrationC0_BackwardPumpTransmissionYValue := 479, txt_DbVar_C0_NvCalibrationC0_BackwardPumpTransmissionYValue_0 := 480, txt_DbVar_C0_NvCalibrationC0_BackwardPumpTransmissionYValue_1 := 481, txt_DbVarArrDescr_C0_NvCalibrationC0_ForwardPumpTransmissionRampRatio := 482, txt_DbVar_C0_NvCalibrationC0_ForwardPumpTransmissionRampRatio_0 := 483, txt_DbVar_C0_NvCalibrationC0_ForwardPumpTransmissionRampRatio_1 := 484, txt_DbVarArrDescr_C0_NvCalibrationC0_RangeValueForwardPumpTransRamp := 485, txt_DbVar_C0_NvCalibrationC0_RangeValueForwardPumpTransRamp_0 := 486, txt_DbVar_C0_NvCalibrationC0_RangeValueForwardPumpTransRamp_1 := 487, txt_DbVar_C0_NvCalibrationC0_RangeValueForwardPumpTransRamp_2 := 488, txt_DbVarArrDescr_C0_NvCalibrationC0_BackwardPumpTransmissionRampRtio := 489, txt_DbVar_C0_NvCalibrationC0_BackwardPumpTransmissionRampRtio_0 := 490, txt_DbVar_C0_NvCalibrationC0_BackwardPumpTransmissionRampRtio_1 := 491, txt_DbVarArrDescr_C0_NvCalibrationC0_RangeValueBackwardPumpTransRamp := 492, txt_DbVar_C0_NvCalibrationC0_RangeValueBackwardPumpTransRamp_0 := 493, txt_DbVar_C0_NvCalibrationC0_RangeValueBackwardPumpTransRamp_1 := 494, txt_DbVar_C0_NvCalibrationC0_RangeValueBackwardPumpTransRamp_2 := 495, txt_DbVar_C0_NvCalibrationC0_EncodeurTurretOffset_0 := 496, txt_DbVar_C0_NvCalibrationC0_SlopeLongOffset_0 := 497, txt_DbVar_C0_NvCalibrationC0_SlopeTransOffset_0 := 498, txt_DbVar_C0_NvCalibrationC0_SlopeLongOffset2_0 := 499, txt_DbVar_C0_NvCalibrationC0_SlopeTransOffset2_0 := 500, txt_DbVar_C0_NvCalibrationC0_EncodeurTurretOffset2_0 := 501, txt_DbVar_C0_NvCalibrationC0_EncodeurTurretMsb1_0 := 502, txt_DbVar_C0_NvCalibrationC0_EncodeurTurretMsb2_0 := 503, txt_DbVar_C0_NvCalibrationC0_EncodeurTurretLsb1_0 := 504, txt_DbVar_C0_NvCalibrationC0_EncodeurTurretLsb2_0 := 505, txt_DbVar_C0_Ram48XsInputsC0_UpInclinaisonBasketButton_0 := 506, txt_DbVar_C0_Ram48XsInputsC0_UpInclinaisonBasketButtonValue_0 := 507, txt_DbVar_C0_Ram48XsInputsC0_DownInclinaisonBasketButton_0 := 508, txt_DbVar_C0_Ram48XsInputsC0_DownInclinaisonBasketButtonValue_0 := 509, txt_DbVar_C0_Ram48XsInputsC0_UpPendularButton_0 := 510, txt_DbVar_C0_Ram48XsInputsC0_UpPendularButtonValue_0 := 511, txt_DbVar_C0_Ram48XsInputsC0_DownPendularButton_0 := 512, txt_DbVar_C0_Ram48XsInputsC0_DownPendularButtonValue_0 := 513, txt_DbVar_C0_Ram48XsInputsC0_RotationCtClockwiseBasketButton_0 := 514, txt_DbVar_C0_Ram48XsInputsC0_RotCtClockwiseBasketButtonVal_0 := 515, txt_DbVar_C0_Ram48XsInputsC0_RotationClockwiseBasketButton_0 := 516, txt_DbVar_C0_Ram48XsInputsC0_RotationClockwiseBasketButtonVal_0 := 517, txt_DbVar_C0_Ram48XsInputsC0_Overload1_0 := 518, txt_DbVar_C0_Ram48XsInputsC0_Overload1Value_0 := 519, txt_DbVar_C0_Ram48XsInputsC0_Overload2_0 := 520, txt_DbVar_C0_Ram48XsInputsC0_Overload2Value_0 := 521, txt_DbVar_C0_Ram48XsInputsC0_NacelleBasketRightSideSensor1_0 := 522, txt_DbVar_C0_Ram48XsInputsC0_NacelleBasketRightSideSensor1Val_0 := 523, txt_DbVar_C0_Ram48XsInputsC0_NacelleBasketRightSideSensor2_0 := 524, txt_DbVar_C0_Ram48XsInputsC0_NacelleBasketRightSideSensor2Val_0 := 525, txt_DbVar_C0_Ram48XsInputsC0_NacelleBasketLeftSideSensor1_0 := 526, txt_DbVar_C0_Ram48XsInputsC0_NacelleBasketLeftSideSensor1Val_0 := 527, txt_DbVar_C0_Ram48XsInputsC0_NacelleBasketLeftSideSensor2_0 := 528, txt_DbVar_C0_Ram48XsInputsC0_NacelleBasketLeftSideSensor2Val_0 := 529, txt_DbVar_C0_Ram48XsInputsC0_LowSectorPendularSensor_0 := 530, txt_DbVar_C0_Ram48XsInputsC0_LowSectorPendularSensorVal_0 := 531, txt_DbVar_C0_Ram48XsInputsC0_HighSectorPlateSensor_0 := 532, txt_DbVar_C0_Ram48XsInputsC0_HighSectorPlateSensorVal_0 := 533, txt_DbVar_C0_Ram48XsInputsC0_FoldedLadderSensor_0 := 534, txt_DbVar_C0_Ram48XsInputsC0_FoldedLadderSensorVal_0 := 535, txt_DbVar_C0_Ram48XsInputsC0_SafetyManSystem_0 := 536, txt_DbVar_C0_Ram48XsInputsC0_DeltaArmAxisJoystick_0 := 537, txt_DbVar_C0_Ram48XsInputsC0_ArrowArmAxisJoystick_0 := 538, txt_DbVar_C0_Ram48XsInputsC0_TelescopeArmAxisJoysitck_0 := 539, txt_DbVar_C0_Ram48XsInputsC0_RotationTurretAxisJoystick_0 := 540, txt_DbVar_C0_Ram48XsInputsC0_AdvanceAxisJoystick_0 := 541, txt_DbVar_C0_Ram48XsInputsC0_RearmementSafetyManSystem_0 := 542, txt_DbVar_C0_Ram48XsInputsC0_RearmementSafetyManSystemVal_0 := 543, txt_DbVar_C0_Ram48XsInputsC0_AbutementNacelleTrackSide_0 := 544, txt_DbVar_C0_Ram48XsInputsC0_AbutementNacelleTrackSideVal_0 := 545, txt_DbVar_C0_Ram48XsInputsC0_AbutementNacelleCenteredSide_0 := 546, txt_DbVar_C0_Ram48XsInputsC0_AbutementNacelleCenteredSideVal_0 := 547, txt_DbVar_C0_Ram48XsInputsC0_DeltaArmJystckCenteredTelescope_0 := 548, txt_DbVar_C0_Ram48XsInputsC0_ArrowJoystickCenteredTurret_0 := 549, txt_DbVar_C0_Ram48XsInputsC0_CenteredAdvanceJoystick_0 := 550, txt_DbVar_C0_Ram48XsInputsC0_DeadManPedal_0 := 551, txt_DbVar_C0_Ram48XsInputsC0_PressenceInNacelleSensor1_0 := 552, txt_DbVar_C0_Ram48XsInputsC0_PressenceInNacelleSensor2_0 := 553, txt_DbVar_C0_Ram48XsInputsC0_Gachette_0 := 554, txt_DbVar_C0_Ram48XsInputsC0_Klaxon_0 := 555, txt_DbVar_C0_Ram48XsInputsC0_StopMotorButton_0 := 556, txt_DbVar_C0_Ram48XsInputsC0_AuthorizationWorkKey_0 := 557, txt_DbVar_C0_Ram48XsInputsC0_EtallonnageJoystickButton_0 := 558, txt_DbVar_C0_Ram48XsInputsC0_ClosePortillonSensor_0 := 559, txt_DbVar_C0_Ram48XsInputsC0_Hearbeat48Xs_0 := 560, txt_DbVar_C0_Ram48XsInputsC0_BatterieVoltage48Xs_0 := 561, txt_DbVar_C0_Ram48XsOutputsC0_WhiteLightsCommand_0 := 562, txt_DbVar_C0_Ram48XsOutputsC0_WhiteLightsValue_0 := 563, txt_DbVar_C0_Ram48XsOutputsC0_RedLightsCommand_0 := 564, txt_DbVar_C0_Ram48XsOutputsC0_RedLightsValue_0 := 565, txt_DbVar_C0_Ram48XsOutputsC0_WorkLightCommand_0 := 566, txt_DbVar_C0_Ram48XsOutputsC0_WorkLightValue_0 := 567, txt_DbVar_C0_Ram48XsOutputsC0_BuzzerCommand_0 := 568, txt_DbVar_C0_Ram48XsOutputsC0_BuzzerValue_0 := 569, txt_DbVar_C0_Ram48XsOutputsC0_MotorDefaultLightErrSta_0 := 570, txt_DbVar_C0_Ram48XsOutputsC0_OverloadLightErrSta_0 := 571, txt_DbVar_C0_Ram48XsOutputsC0_BuzzerErrSta_0 := 572, txt_DbVar_C0_Ram48XsOutputsC0_GasOilLightErrSta_0 := 573, txt_DbVar_C0_Ram48XsOutputsC0_DeversDefaultLightErrSta_0 := 574, txt_DbVar_C0_Ram48XsOutputsC0_RedLightARDErrSta_0 := 575, txt_DbVar_C0_Ram48XsOutputsC0_WhiteLightARDErrSta_0 := 576, txt_DbVar_C0_Ram48XsOutputsC0_WarmingLightErrSta_0 := 577, txt_DbVar_C0_Ram48XsOutputsC0_RedLightARGErrSta_0 := 578, txt_DbVar_C0_Ram48XsOutputsC0_WhiteLightARGErrSta_0 := 579, txt_DbVar_C0_RamEcuInputRadioControl_StateRadioControl_0 := 580, txt_DbVar_C0_RamEcuInputRadioControl_LeftManipulator_0 := 581, txt_DbVar_C0_RamEcuInputRadioControl_RightManipulator_0 := 582, txt_DbVar_C0_RamEcuInputRadioControl_LeftManipulatorPosition_0 := 583, txt_DbVar_C0_RamEcuInputRadioControl_RightManipulatorPosition_0 := 584, txt_DbVar_C0_RamEcuInputRadioControl_UpAxleArFixe_0 := 585, txt_DbVar_C0_RamEcuInputRadioControl_DownAxleArFixe_0 := 586, txt_DbVar_C0_RamEcuInputRadioControl_UpAxleAvOscillant_0 := 587, txt_DbVar_C0_RamEcuInputRadioControl_DownAxleAvOscillant_0 := 588, txt_DbVar_C0_RamEcuInputRadioControl_RotationFrameCtClkwise_0 := 589, txt_DbVar_C0_RamEcuInputRadioControl_RotationFrameClkwise_0 := 590, txt_DbVar_C0_RamEcuInputRadioControl_SelectorRotTurret_0 := 591, txt_DbVar_C0_RamEcuInputRadioControl_SelectorPendular_0 := 592, txt_DbVar_C0_RamEcuInputRadioControl_RadioCommandConnect_0 := 593, txt_DbVar_C0_RamEcuInputRadioControl_UpPendularOrRotCtClkTurret_0 := 594, txt_DbVar_C0_RamEcuInputRadioControl_DownPendularOrRotClkTurret_0 := 595, txt_DbVar_C0_RamEcuInputRadioControl_StartRadioCommand_0 := 596, txt_DbVar_C0_RamEcuInputRadioControl_StopRadioCommand_0 := 597, txt_DbVar_C0_RamEcuInputRadioControl_ForcingAdvanceTrack_0 := 598, txt_DbVar_C0_RamEcuInputRadioControl_KlaxonCommand_0 := 599, txt_DbVar_C0_RamCanSensorC0_EncodeurTurret1AngleRaw_0 := 600, txt_DbVar_C0_RamCanSensorC0_EncodeurTurret1Angle_0 := 601, txt_DbVar_C0_RamCanSensorC0_EncodeurTurret2AngleRaw_0 := 602, txt_DbVar_C0_RamCanSensorC0_EncodeurTurret2Angle_0 := 603, txt_DbVar_C0_RamCanSensorC0_SlopeLongAngleSensor1_0 := 604, txt_DbVar_C0_RamCanSensorC0_SlopeTransAngleSensor1_0 := 605, txt_DbVar_C0_RamCanSensorC0_SlopeLongAngleValue_0 := 606, txt_DbVar_C0_RamCanSensorC0_SlopeTransAngleValue_0 := 607, txt_DbVar_C0_RamCanSensorC0_StateHeartBeatDeversSensor_0 := 608, txt_DbVar_C0_RamCanSensorC0_StateHeartBeatEncodeurTurret1_0 := 609, txt_DbVar_C0_RamCanSensorC0_SelectedSlopeAngle_0 := 610, txt_DbVar_C0_RamCanSensorC0_EncodeurMastMeasureRaw_0 := 611, txt_DbVar_C0_RamCanSensorC0_EncodeurMastMeasureCentimeter_0 := 612, txt_DbVar_C0_RamCanSensorC0_SlopeLongAngleSensor2_0 := 613, txt_DbVar_C0_RamCanSensorC0_SlopeTransAngleSensor2_0 := 614, txt_DbVar_C0_RamCanSensorC0_SlopeAlarm1_0 := 615, txt_DbVar_C0_RamCanSensorC0_SlopeAlarm2_0 := 616, txt_DbVar_C0_RamCanSensorC0_SlopeLongAngleValue2_0 := 617, txt_DbVar_C0_RamCanSensorC0_SlopeTransAngleValue2_0 := 618, txt_DbVar_C0_RamCanSensorC0_ErrorCodeEncodeurTurret1_0 := 619, txt_DbVar_C0_RamCanSensorC0_ErrorRegisterEncodeurTurret1_0 := 620, txt_DbVar_C0_RamCanSensorC0_ErrorCodeEncodeurTurret2_0 := 621, txt_DbVar_C0_RamCanSensorC0_ErrorRegisterEncodeurTurret2_0 := 622, txt_DbVar_C0_RamCanSensorC0_ErrorCodeMastMeasure_0 := 623, txt_DbVar_C0_RamCanSensorC0_ErrorRegisterMastMeasure_0 := 624, txt_DbVar_C0_RamCanSensorC0_StateHeartBeatDeversSensor2_0 := 625, txt_DbVar_C0_RamCanSensorC0_TimeoutSdoReqDetectedEncdTurret1_0 := 626, txt_DbVar_C0_RamCanSensorC0_TimeoutSdoReqDetectedEncdTurret2_0 := 627, txt_DbVar_C0_RamCanSensorC0_EncodeurTurretOffset_0 := 628, txt_DbVar_C0_RamCanSensorC0_EncodeurTurretOffset2_0 := 629, txt_DbVar_C0_RamEvision7C0_LoginStatus_0 := 630, txt_DbVar_C0_RamEvision7C0_AllowMovementNacelle_0 := 631, txt_DbVar_C0_RamEvision7C0_gBreak_Parking_On_Off_0 := 632, txt_DbVar_C0_RamEvision7C0_gBreak_Faillure_On_Off_0 := 633, txt_DbVar_C0_RamEvision7C0_gTurretInCenter_0 := 634, txt_DbVar_C0_RamEvision7C0_gTurretSectorInCenter_0 := 635, txt_DbVar_C0_RamEvision7C0_gVehiculeTrainMode_0 := 636, txt_DbVar_C0_RamEvision7C0_gIncoherenceLateralStopAndKey_0 := 637, txt_DbVar_C0_RamEvision7C0_gWorkMode_0 := 638, txt_DbVar_C0_RamEvision7C0_gSafetyElectricPump_0 := 639, txt_DbVar_C0_RamEvision7C0_gDownhill150mm_0 := 640, txt_DbVar_C0_RamEvision7C0_gTrainModeAllow_0 := 641, txt_DbVar_C0_RamEvision7C0_gBrakeTestService_0 := 642, txt_DbVar_C0_RamEvision7C0_gBrakePressureFault_0 := 643, txt_DbVar_C0_RamEvision7C0_gActivateMeasuringMast_0 := 644, txt_DbVar_C0_RamEvision7C0_gAutoMovementDirectionLight_0 := 645, txt_DbVar_C0_RamEvision7C0_gBackRailwayAxleLowPosition_0 := 646, txt_DbVar_C0_RamEvision7C0_gFrontRailwayAxleLowPosition_0 := 647, txt_DbVar_C0_RamEvision7C0_gBackRailwayAxleServiceBrake_0 := 648, txt_DbVar_C0_RamEvision7C0_gFrontRailwayAxleServiceBrake_0 := 649, txt_DbVar_C0_RamEvision7C0_gBackRailwayAxleParkBrake_0 := 650, txt_DbVar_C0_RamEvision7C0_gFrontRailwayAxleParkBrake_0 := 651, txt_DbVar_C0_RamEvision7C0_gStatusFrontLeftTrainBrakeTest_0 := 652, txt_DbVar_C0_RamEvision7C0_gStatusFrontRightTrainBrakeTest_0 := 653, txt_DbVar_C0_RamEvision7C0_gStatusBackLeftTrainBrakeTest_0 := 654, txt_DbVar_C0_RamEvision7C0_gStatusBackRightTrainBrakeTest_0 := 655, txt_DbVar_C0_RamEvision7C0_gAlarmAru_0 := 656, txt_DbVar_C0_RamEvision7C0_gEngine_Use_Time_0 := 657, txt_DbVar_C0_RamEvision7C0_gEngine_RPM_0 := 658, txt_DbVar_C0_RamEvision7C0_gVehiculeSpeed_0 := 659, txt_DbVar_C0_RamEvision7C0_gLateralizationStop_0 := 660, txt_DbVar_C0_RamEvision7C0_gKeySelector_0 := 661, txt_DbVar_C0_RamEvision7C0_gFrontSpeedRailWayAxle_0 := 662, txt_DbVar_C0_RamEvision7C0_gBackSpeedRailWayAxle_0 := 663, txt_DbVar_C0_RamEvision7C0_gButtonCalibTurretEncoder_0 := 664, txt_DbVar_C0_RamEvision7C0_gOffTrackTestBrakeActivated_0 := 665, txt_DbVar_C0_RamEvision7C0_gOffTrackRunInBrakeActivated_0 := 666, txt_DbVar_C0_RamEvision7C0_gOsciServiceBrakeSelect_0 := 667, txt_DbVar_C0_RamEvision7C0_gFixedServiceBrakeSelect_0 := 668, txt_DbVar_C0_RamEvision7C0_gBothServiceBrakeSelect_0 := 669, txt_DbVar_C0_RamEvision7C0_gOsciParkBrakeSelect_0 := 670, txt_DbVar_C0_RamEvision7C0_gFixedParkBrakeSelect_0 := 671, txt_DbVar_C0_RamEvision7C0_gBothParkBrakeSelect_0 := 672, txt_DbVar_C0_RamEvision7C0_gOsciServiceRunInBrakeSelect_0 := 673, txt_DbVar_C0_RamEvision7C0_gFixedServiceRunInBrakeSelect_0 := 674, txt_DbVar_C0_RamEvision7C0_gBothServiceRunInBrakeSelect_0 := 675, txt_DbVar_C0_RamEvision7C0_gTestBrakePageActive_0 := 676, txt_DbVar_C0_RamEvision7C0_gBreakInBrakePageActive_0 := 677, txt_DbVar_C0_RamEvision7C0_gSerialNumber_0 := 678, txt_DbVar_C0_RamEvision7C0_gBPBasketValidate_0 := 679, txt_DbVar_C0_RamEvision7C0_gKeyFilterOverload_0 := 680, txt_DbVar_C0_RamEvision7C0_gKeyNextMode_0 := 681, txt_DbVar_C0_RamEvision7C0_gKeyPrevMode_0 := 682, txt_DbVar_C0_RamEvision7C0_gKeySignalDanger_0 := 683, txt_DbVar_C0_RamEvision7C0_gKeyFlashLightON_0 := 684, txt_DbVar_C0_RamEvision7C0_gKeyCalibMastMin_0 := 685, txt_DbVar_C0_RamEvision7C0_gKeyCalibMastMax_0 := 686, txt_DbVar_C0_RamEvision7C0_gKeyCalibMastValid_0 := 687, txt_DbVar_C0_RamEvision7C0_gKeyGeneratorActivate_0 := 688, txt_DbVar_C0_RamEvision7C0_gRazDistanceTraveledMastMeasure_0 := 689, txt_DbVar_C0_RamEvision7C0_gKeyWhiteLights15746_0 := 690, txt_DbVar_C0_RamEvision7C0_gOsci2ndParkBrakeSelect_0 := 691, txt_DbVar_C0_RamEvision7C0_gFixe2ndParkBrakeSelect_0 := 692, txt_DbVar_C0_RamEvision7C0_gKeyRazController_0 := 693, txt_DbVar_C0_RamEcuC0RcvFromC1_C1TurretPostSelector_0 := 694, txt_DbVar_C0_RamEcuC0RcvFromC1_C1RadioPostSelector_0 := 695, txt_DbVar_C0_RamEcuC0RcvFromC1_C1NacellePostSelector_0 := 696, txt_DbVar_C0_RamEcuC0RcvFromC1_UpAxleOscillantCommand_0 := 697, txt_DbVar_C0_RamEcuC0RcvFromC1_DownAxleOscillantCommand_0 := 698, txt_DbVar_C0_RamEcuC0RcvFromC1_UpAxleFixeCommand_0 := 699, txt_DbVar_C0_RamEcuC0RcvFromC1_DownAxleFixeCommand_0 := 700, txt_DbVar_C0_RamEcuC0RcvFromC1_RegimeMotorAlternatorRpm_0 := 701, txt_DbVar_C0_RamEcuC0RcvFromC1_EntryTelescopeFdcSensor_0 := 702, txt_DbVar_C0_RamEcuC0RcvFromC1_DeltaArmFoldedSensor_0 := 703, txt_DbVar_C0_RamEcuC0RcvFromC1_BoomArmFoldedSensor_0 := 704, txt_DbVar_C0_RamEcuC0RcvFromC1_DeltaArmInLowerZone_0 := 705, txt_DbVar_C0_RamEcuC0RcvFromC1_ArrowArmAngularSensor_0 := 706, txt_DbVar_C0_RamEcuC0RcvFromC1_TurretInRearCenterPos_0 := 707, txt_DbVar_C0_RamEcuC0RcvFromC1_TurretInFrontCenterPos_0 := 708, txt_DbVar_C0_RamEcuC0RcvFromC1_FoldedDeltaArmZone_0 := 709, txt_DbVar_C0_RamEcuC0RcvFromC1_FoldedArrowArmZone_0 := 710, txt_DbVar_C0_RamEcuC0RcvFromC1_NoMovementIsDuring_0 := 711, txt_DbVar_C0_RamEcuC0RcvFromC1_DeltaArmAngularSensor_0 := 712, txt_DbVar_C0_RamEcuC0RcvFromC1_FoldedMastMeasure_0 := 713, txt_DbVar_C0_RamEcuC0RcvFromC1_Transmission1Pressure_0 := 714, txt_DbVar_C0_RamEcuC0RcvFromC1_Transmission2Pressure_0 := 715, txt_DbVar_C0_RamEcuC0RcvFromC1_ActiveHelpState_0 := 716, txt_DbVar_C0_RamEcuC0RcvFromC1_BasketInCentrerPos_0 := 717, txt_DbVar_C0_RamEcuC0RcvFromC1_StopAllMovementsNacellePost_0 := 718, txt_DbVar_C0_RamEcuC0RcvFromC1_EncodeurMastMeasureCentimeter_0 := 719, txt_DbVar_C0_RamEcuC0RcvFromC1_MastMeasureFonctionActive_0 := 720, txt_DbVar_C0_RamEcuC0RcvFromC1_OutOfRangeTransmissionPressure_0 := 721, txt_DbVar_C0_RamEcuC0RcvFromC1_Beacon_0 := 722, txt_DbVar_C0_RamEcuC0RcvFromC1_MotorOn_0 := 723, txt_DbVar_C0_RamEcuC0RcvFromC1_FaultLenghtSensor_0 := 724, txt_DbVar_C0_RamEcuC0RcvFromC1_TurretSensorsFailures_0 := 725, txt_DbVar_C0_RamEcuC0RcvFromC1_OptionWhiteLight15746_0 := 726, txt_DbVar_C0_RamEcuC0RcvFromC1_SafeManSystem_0 := 727, txt_DbVar_C0_RamEcuC0RcvFromC1_SlopeModeFromC1_0 := 728, txt_DbVar_C0_RamEcuC0RcvFromC1_ColdOilTankTemperature_0 := 729, txt_DbVar_C0_RamEcuC0RcvFromC1_ElectricMotorForbidden_0 := 730, txt_DbVar_C0_RamEcuC0RcvFromC1_RpmMotorElectric_0 := 731, txt_DbVar_C0_RamEcuC0RcvFromC1_OilTankTemperatureValue_0 := 732, txt_DbVar_C0_RamEcuC0RcvFromC1_SocStopRegen_0 := 733, txt_DbVar_C0_RamEcuC0RcvFromC1_GeneratorOn_0 := 734, txt_DbVar_C0_RamEcuC0RcvFromC1_EvDevMvtsCmd_0 := 735, txt_DbVar_C0_RamEcuC0RcvFromC1_TestElectricalFromC1_0 := 736, txt_DbVar_C0_RamEcuC0RcvFromC1_AutoModeActivate_0 := 737, txt_DbVar_C0_RamEcuC0RcvFromC1_SilenceModeActivate_0 := 738, txt_DbVar_C0_RamEcuC0RcvFromC1_ForcingRegenlow_0 := 739, txt_DbVar_C0_RamEcuC0RcvFromC1_ForcingRegenHigh_0 := 740, txt_DbVar_C0_RamEcuC0RcvFromC1_EvBypassCommand_0 := 741, txt_DbVar_C0_RamEcuC0RcvFromC1_MotorspeedCmdJ1939_0 := 742, txt_DbVar_C0_RamEcuCaliCmdC0_CalibTurretAngle_0 := 743, txt_DbVar_C0_RamEcuCaliCmdC0_CalibTurretAngleIntermedaireBool_0 := 744, txt_DbVar_C0_RamEcuCaliCmdC0_CalibSlopeLong_0 := 745, txt_DbVar_C0_RamEcuCaliCmdC0_CalibSlopeTrans_0 := 746, txt_DbVar_C0_RamEcuCaliCmdC0_SavedCalibrationListC0_0 := 747, txt_DbVar_C0_NvParamSpeedMaxRail_AccesSiteSpeedForward_0 := 748, txt_DbVar_C0_NvParamSpeedMaxRail_HighSpeedForward_0 := 749, txt_DbVar_C0_NvParamSpeedMaxRail_LowSpeedForward_0 := 750, txt_DbVar_C0_NvParamSpeedMaxRail_LowSpeedBrakeTestForward_0 := 751, txt_DbVar_C0_NvParamSpeedMaxRail_HighSpeedSlopeTresholdAbs_0 := 752, txt_DbVar_C0_NvParamSpeedMaxRail_HighSpeedSlopeTresholdHystRel_0 := 753, txt_DbVar_C0_NvParamSpeedMaxRail_LowSpeedSlopeTresholdAbs_0 := 754, txt_DbVar_C0_NvParamSpeedMaxRail_LowSpeedSlopeTresholdHystRel_0 := 755, txt_DbVar_C0_NvParamSpeedMaxRail_TurretLowSpeedTresholdRel_0 := 756, txt_DbVar_C0_NvParamSpeedMaxRail_TurretLowSpeedTresholdHyst_0 := 757, txt_DbVar_C0_NvParamSpeedMaxRail_TurretRearCenterPos_0 := 758, txt_DbVar_C0_NvParamSpeedMaxRail_TurretFrontPositiveCenterPos_0 := 759, txt_DbVar_C0_NvParamSpeedMaxRail_TurretFrontNegativeCenterPos_0 := 760, txt_DbVar_C0_NvParamSpeedMaxRail_LimitSpeedAccesSiteSpeed_0 := 761, txt_DbVar_C0_NvParamSpeedMaxRail_LimitSpeedHighSpeed_0 := 762, txt_DbVar_C0_NvParamSpeedMaxRail_LimitSpeedLowSpeed_0 := 763, txt_DbVar_C0_NvParamSpeedMaxRail_LimitSpeedLowSpeedBrakeTest_0 := 764, txt_DbVar_C0_NvParamSpeedMaxRail_AccesSiteSpeedBackward_0 := 765, txt_DbVar_C0_NvParamSpeedMaxRail_HighSpeedBackward_0 := 766, txt_DbVar_C0_NvParamSpeedMaxRail_LowSpeedBackward_0 := 767, txt_DbVar_C0_NvParamSpeedMaxRail_LowSpeedBrakeTestBackward_0 := 768, txt_DbVar_C0_NvParamSpeedMaxRail_TestBrakeSpeedForward_0 := 769, txt_DbVar_C0_NvParamSpeedMaxRail_TestBrakeSpeedBackward_0 := 770, txt_DbVar_C0_NvParamSpeedMaxRail_BreakeInBrakeSpeedForward_0 := 771, txt_DbVar_C0_NvParamSpeedMaxRail_BreakeInBrakeSpeedBackward_0 := 772, txt_DbVar_C0_NvParamSpeedMaxRail_ArmSpeedRailHyst_0 := 773, txt_DbVar_C0_NvParamSpeedMaxRail_ArmLowSectorBasketFaultThres_0 := 774, txt_DbVar_C0_NvParamSpeedMaxRail_ArmLowZoneForLowSpeed_0 := 775, txt_DbVar_C0_NvParamSpeedMaxRail_TurretRearNegLowSpeedTreshold_0 := 776, txt_DbVar_C0_NvParamSpeedMaxRail_TurretRearPosLowSpeedTreshold_0 := 777, txt_DbVar_C0_NvParamSpeedMaxRail_Performance2DegSlopeThres_0 := 778, txt_DbVar_C0_NvParamSpeedMaxRail_Performance4DegSlopeThres_0 := 779, txt_DbVar_C0_NvParamSpeedMaxRail_Performance6DegSlopeThres_0 := 780, txt_DbVar_C0_NvParamSpeedMaxRail_PerformanceDegSlopeHyst_0 := 781, txt_DbVar_C0_NvParamSpeedMaxRail_TurretPerfLowSpeedHystHigh_0 := 782, txt_DbVar_C0_NvParamSpeedMaxRail_TurretPerformLowSpeed2Deg_0 := 783, txt_DbVar_C0_NvParamSpeedMaxRail_TurretPerformLowSpeedBasketRot2_0 := 784, txt_DbVar_C0_NvParamSpeedMaxRail_TurretPerformLowSpeed4Deg_0 := 785, txt_DbVar_C0_NvParamSpeedMaxRail_TurretPerfLowSpeedBasketRot4Deg_0 := 786, txt_DbVar_C0_NvParamSpeedMaxRail_TurretPerformLowSpeed6Deg_0 := 787, txt_DbVar_C0_NvParamSpeedMaxRail_TurretPerfLowSpeedBasketRot6Deg_0 := 788, txt_DbVar_C0_NvParamSpeedMaxRail_PreventLimitSpeedAccesSiteSpeed_0 := 789, txt_DbVar_C0_NvParamSpeedMaxRail_PreventLimitSpeedHighSpeed_0 := 790, txt_DbVar_C0_NvParamSpeedMaxRail_PreventLimitSpeedLowSpeed_0 := 791, txt_DbVar_C0_NvParamSpeedMaxRail_PreventSpeedLowSpeedBrakeTest_0 := 792, txt_DbVar_C0_RamSpeedMaxRail_SlopeOverHighSpeedTresh_0 := 793, txt_DbVar_C0_RamSpeedMaxRail_SlopeLowerLowSpeedTresh_0 := 794, txt_DbVar_C0_RamSpeedMaxRail_TurretInLowSpeedRearZone_0 := 795, txt_DbVar_C0_RamSpeedMaxRail_TurretInLowSpeedPosFrontZone_0 := 796, txt_DbVar_C0_RamSpeedMaxRail_TurretInLowSpeedNegFrontZone_0 := 797, txt_DbVar_C0_RamSpeedMaxRail_TurretInLowSpeedZone_0 := 798, txt_DbVar_C0_RamSpeedMaxRail_EnableSimuMode_0 := 799, txt_DbVar_C0_RamSpeedMaxRail_SimuDevers_0 := 800, txt_DbVar_C0_RamSpeedMaxRail_SimuTurretAngle_0 := 801, txt_DbVar_C0_RamSpeedMaxRail_SimuAuthorizationWorkKey_0 := 802, txt_DbVar_C0_RamSpeedMaxRail_SimuAbutmentTurretCentred_0 := 803, txt_DbVar_C0_RamSpeedMaxRail_SimuWorkKeyCentred_0 := 804, txt_DbVar_C0_RamSpeedMaxRail_SimuTelescopeEntry_0 := 805, txt_DbVar_C0_RamSpeedMaxRail_SimuDeltaArmFoldedSensor_0 := 806, txt_DbVar_C0_RamSpeedMaxRail_SimuDeltaArmFoldedZone_0 := 807, txt_DbVar_C0_RamSpeedMaxRail_SimuArrowArmFoldedSensor_0 := 808, txt_DbVar_C0_RamSpeedMaxRail_SimuArrowArmFoldedZone_0 := 809, txt_DbVar_C0_RamSpeedMaxRail_SimuNacelleBasketLeftSideSensor1_0 := 810, txt_DbVar_C0_RamSpeedMaxRail_SimuNacelleBasketLeftSideSensor2_0 := 811, txt_DbVar_C0_RamSpeedMaxRail_SimuNacelleBasketRighSideSensor1_0 := 812, txt_DbVar_C0_RamSpeedMaxRail_SimuNacelleBasketRighSideSensor2_0 := 813, txt_DbVar_C0_RamSpeedMaxRail_SimuHighSectorPlateSensor_0 := 814, txt_DbVar_C0_RamSpeedMaxRail_RailSpeedMaxMode_0 := 815, txt_DbVar_C0_RamSpeedMaxRail_SimuDeltaArmInLowerZone_0 := 816, txt_DbVar_C0_RamSpeedMaxRail_SimuTurretInRearCenterPos_0 := 817, txt_DbVar_C0_RamSpeedMaxRail_SimuTurretInFrontCenterPos_0 := 818, txt_DbVar_C0_RamSpeedMaxRail_LimitSpeedAccesSiteSpeedExceeded_0 := 819, txt_DbVar_C0_RamSpeedMaxRail_LimitSpeedHighSpeedExceeded_0 := 820, txt_DbVar_C0_RamSpeedMaxRail_LimitSpeedLowSpeedExceeded_0 := 821, txt_DbVar_C0_RamSpeedMaxRail_LimitSpeedLowSpeedBrakeTestExced_0 := 822, txt_DbVar_C0_RamSpeedMaxRail_LitmitSpeedExceeded_0 := 823, txt_DbVar_C0_RamSpeedMaxRail_KinematicTrainAllow_0 := 824, txt_DbVar_C0_RamSpeedMaxRail_SlopeCaseLess2Deg_0 := 825, txt_DbVar_C0_RamSpeedMaxRail_SlopeCaseLess4Deg_0 := 826, txt_DbVar_C0_RamSpeedMaxRail_SlopeCaseLess6Deg_0 := 827, txt_DbVar_C0_RamSpeedMaxRail_SlopeCaseHigher6Deg_0 := 828, txt_DbVar_C0_RamSpeedMaxRail_TurretInSpeedZone2Deg_0 := 829, txt_DbVar_C0_RamSpeedMaxRail_TurretInSpeedZone4Deg_0 := 830, txt_DbVar_C0_RamSpeedMaxRail_TurretInSpeedZone6Deg_0 := 831, txt_DbVar_C0_RamSpeedMaxRail_TurretInSpeedZone2DegForBasket_0 := 832, txt_DbVar_C0_RamSpeedMaxRail_TurretInSpeedZone4DegForBasket_0 := 833, txt_DbVar_C0_RamSpeedMaxRail_TurretInSpeedZone6DegForBasket_0 := 834, txt_DbVar_C0_RamSpeedMaxRail_PreventLimitSpeedAccesSiteSpeed_0 := 835, txt_DbVar_C0_RamSpeedMaxRail_PreventLimitSpeedHighSpeed_0 := 836, txt_DbVar_C0_RamSpeedMaxRail_PreventLimitSpeedLowSpeed_0 := 837, txt_DbVar_C0_RamSpeedMaxRail_PreventLimitLowSpeedBrakeTest_0 := 838, txt_DbVar_C0_RamSpeedMaxRail_PreventLimitSpeedExceeding_0 := 839, txt_DbVar_C0_RamSpeedMaxRail_AuthoriseGlobalLowSpeed_0 := 840, txt_DbVar_C0_NvParamBrakeTest_NCycleNeedBrakeTest_0 := 841, txt_DbVar_C0_NvParamBrakeTest_NCyclesBrakeCritical_0 := 842, txt_DbVar_C0_NvParamBrakeTest_SpeedMinTreshIncrBrakeCycles_0 := 843, txt_DbVar_C0_NvParamBrakeTest_PressureOsciServiceBrakeTresh_0 := 844, txt_DbVar_C0_NvParamBrakeTest_PressureFixeServiceBrakeTresh_0 := 845, txt_DbVar_C0_NvParamBrakeTest_PressureOsciParkingBrakeTresh_0 := 846, txt_DbVar_C0_NvParamBrakeTest_PressureFixeParkingBrakeTresh_0 := 847, txt_DbVar_C0_NvParamBrakeTest_TimeOsciSerivceBrakeMs_0 := 848, txt_DbVar_C0_NvParamBrakeTest_TimeFixeSerivceBrakeMs_0 := 849, txt_DbVar_C0_NvParamBrakeTest_TimeOsciParkingBrakeMs_0 := 850, txt_DbVar_C0_NvParamBrakeTest_TimeFixeParkingBrakeMs_0 := 851, txt_DbVar_C0_NvParamBrakeTest_SpeedMinBrakeTestRunning_0 := 852, txt_DbVar_C0_NvParamBrakeTest_ValidCondiEnableTestBrakeTime_0 := 853, txt_DbVar_C0_NvParamBrakeTest_NbElementDeltaTransmPressure_0 := 854, txt_DbVar_C0_NvParamBrakeTest_NCycleNeed2ndParkBrake_0 := 855, txt_DbVar_C0_NvParamBrakeTest_NCycles2ndBrakeCritical_0 := 856, txt_DbVar_C0_NvParamBrakeTest_TimeOsci2ndParkingBrakeMs_0 := 857, txt_DbVar_C0_NvParamBrakeTest_TimeFixe2ndParkingBrakeMs_0 := 858, txt_DbVar_C0_NvParamBrakeTest_ThresCpt2ndParkBrake_0 := 859, txt_DbVar_C0_NvParamBrakeTest_MinThresholdActive2ndParkBrake_0 := 860, txt_DbVar_C0_RamBrakeTest_ForbidCameraDisplay_0 := 861, txt_DbVar_C0_RamBrakeTest_PressureEfficiencyRate_0 := 862, txt_DbVar_C0_RamBrakeTest_BrakeTestSelected_0 := 863, txt_DbVar_C0_RamBrakeTest_NeedTestBrake_0 := 864, txt_DbVar_C0_RamBrakeTest_CycleBrakeOverCriticalNumber_0 := 865, txt_DbVar_C0_RamBrakeTest_UpPositionAxles_0 := 866, txt_DbVar_C0_RamBrakeTest_DownPositionAxles_0 := 867, txt_DbVar_C0_RamBrakeTest_IncoherencePosAxleAndTestMode_0 := 868, txt_DbVar_C0_RamBrakeTest_TestBrakeInOffrailMode_0 := 869, txt_DbVar_C0_RamBrakeTest_BrakeTestRunning_0 := 870, txt_DbVar_C0_RamBrakeTest_ValidBrakeTest_0 := 871, txt_DbVar_C0_RamBrakeTest_EnableIncrementCycleBrakePerform_0 := 872, txt_DbVar_C0_RamBrakeTest_ValidOsciServiceBrakeTest_0 := 873, txt_DbVar_C0_RamBrakeTest_ValidFixeServiceBrakeTest_0 := 874, txt_DbVar_C0_RamBrakeTest_ValidOsciParkingBrakeTest_0 := 875, txt_DbVar_C0_RamBrakeTest_ValidFixeParkingBrakeTest_0 := 876, txt_DbVar_C0_RamBrakeTest_SimuOsciServiceBrakeSelect_0 := 877, txt_DbVar_C0_RamBrakeTest_SimuFixeServiceBrakeSelect_0 := 878, txt_DbVar_C0_RamBrakeTest_SimuOsciParkBrakeSelect_0 := 879, txt_DbVar_C0_RamBrakeTest_SimuFixeParkBrakeSelect_0 := 880, txt_DbVar_C0_RamBrakeTest_Simu2ServiceBrakesSelect_0 := 881, txt_DbVar_C0_RamBrakeTest_Simu2ParkBrakesSelect_0 := 882, txt_DbVar_C0_RamBrakeTest_RetainPosJoyAdvance_0 := 883, txt_DbVar_C0_RamBrakeTest_AcutalPosJoyAdvance_0 := 884, txt_DbVar_C0_RamBrakeTest_ForceOsciServiceBrake_0 := 885, txt_DbVar_C0_RamBrakeTest_ForceFixeServiceBrake_0 := 886, txt_DbVar_C0_RamBrakeTest_ForceOsciParkBrake_0 := 887, txt_DbVar_C0_RamBrakeTest_ForceFixeParkBrake_0 := 888, txt_DbVar_C0_RamBrakeTest_StopMovementByBrakeTest_0 := 889, txt_DbVar_C0_RamBrakeTest_AuthorizeTransaltionRail_0 := 890, txt_DbVar_C0_RamBrakeTest_DeltaTransmissionPressure_0 := 891, txt_DbVar_C0_RamBrakeTest_ValidConditionEnableTestBrake_0 := 892, txt_DbVar_C0_RamBrakeTest_TimeOutValidCondition_0 := 893, txt_DbVar_C0_RamBrakeTest_PourcentCycleBrake_0 := 894, txt_DbVar_C0_RamBrakeTest_Force2ndParkBrakeFixe_0 := 895, txt_DbVar_C0_RamBrakeTest_Force2ndParkBrakeOsci_0 := 896, txt_DbVar_C0_RamBrakeTest_ValidOsci2ndParkBrakeTest_0 := 897, txt_DbVar_C0_RamBrakeTest_ValidFixe2ndParkBrakeTest_0 := 898, txt_DbVar_C0_RamBrakeTest_PourcentCycle2ndParkBrake_0 := 899, txt_DbVar_C0_RamBrakeTest_NeedTest2ndParkBrake_0 := 900, txt_DbVar_C0_RamBrakeTest_Cycle2ndParkBrakeCritical_0 := 901, txt_DbVar_C0_RamBrakeTest_AddParkBrakeActive_0 := 902, txt_DbVar_C0_RamBrakeTest_ParkBrake2ndPressureActive_0 := 903, txt_DbVar_C0_NvParamRailWorkSafetyC0_MinTurretAngleConsistALO_0 := 904, txt_DbVar_C0_NvParamRailWorkSafetyC0_MaxTurretAngleConsistALO_0 := 905, txt_DbVar_C0_NvParamRailWorkSafetyC0_MinTurretAngleConsistMultilane_0 := 906, txt_DbVar_C0_NvParamRailWorkSafetyC0_MaxTurretAngleConsistMultilane_0 := 907, txt_DbVar_C0_NvParamRailWorkSafetyC0_ALOTurretRearZoneThres_0 := 908, txt_DbVar_C0_NvParamRailWorkSafetyC0_ALOTurretRearZoneHyst_0 := 909, txt_DbVar_C0_NvParamRailWorkSafetyC0_ALOTurretRearZoneSlowThres_0 := 910, txt_DbVar_C0_NvParamRailWorkSafetyC0_ALOTurretFrontZoneThres_0 := 911, txt_DbVar_C0_NvParamRailWorkSafetyC0_ALOTurretFrontZoneHyst_0 := 912, txt_DbVar_C0_NvParamRailWorkSafetyC0_ALOTurretFrontZoneSlowThres_0 := 913, txt_DbVar_C0_NvParamRailWorkSafetyC0_ALOArrowLowerZoneThres_0 := 914, txt_DbVar_C0_NvParamRailWorkSafetyC0_ALOArrowLowerZoneHyst_0 := 915, txt_DbVar_C0_NvParamRailWorkSafetyC0_ALOArrowLowerZoneSlowThres_0 := 916, txt_DbVar_C0_NvParamRailWorkSafetyC0_ALOTurretRearEndStopThres_0 := 917, txt_DbVar_C0_NvParamRailWorkSafetyC0_ALOTurretRearEndStopHyst_0 := 918, txt_DbVar_C0_NvParamRailWorkSafetyC0_ALOTurretRearEndStopSlowThres_0 := 919, txt_DbVar_C0_NvParamRailWorkSafetyC0_ALOTurretFrontEndStopThres_0 := 920, txt_DbVar_C0_NvParamRailWorkSafetyC0_ALOTurretFrontEndStopHyst_0 := 921, txt_DbVar_C0_NvParamRailWorkSafetyC0_ALOTurretFrontEndStopSlowThres_0 := 922, txt_DbVar_C0_NvParamRailWorkSafetyC0_ALOTurretRearZoneStopThres_0 := 923, txt_DbVar_C0_NvParamRailWorkSafetyC0_ALOTurretRearZoneStopHyst_0 := 924, txt_DbVar_C0_NvParamRailWorkSafetyC0_ALOTurretFrontZoneStopThres_0 := 925, txt_DbVar_C0_NvParamRailWorkSafetyC0_ALOTurretFrontZoneStopHyst_0 := 926, txt_DbVar_C0_NvParamRailWorkSafetyC0_ALOArrowLowerZoneStopThres_0 := 927, txt_DbVar_C0_NvParamRailWorkSafetyC0_ALOArrowLowerZoneStopHyst_0 := 928, txt_DbVar_C0_RamRailWorkSafetyC0_RailWorkMode_0 := 929, txt_DbVar_C0_RamRailWorkSafetyC0_WrongTurretAbutBilateralMode_0 := 930, txt_DbVar_C0_RamRailWorkSafetyC0_WrongTurretAbutMultilaneMode_0 := 931, txt_DbVar_C0_RamRailWorkSafetyC0_WrongTurretAbutALOMode_0 := 932, txt_DbVar_C0_RamRailWorkSafetyC0_WrongBasketAbutBilateralMode_0 := 933, txt_DbVar_C0_RamRailWorkSafetyC0_WrongBasketAbutMultilaneMode_0 := 934, txt_DbVar_C0_RamRailWorkSafetyC0_WrongBasketAbutALOMode_0 := 935, txt_DbVar_C0_RamRailWorkSafetyC0_WrongAbutments_0 := 936, txt_DbVar_C0_RamRailWorkSafetyC0_WrongTurretPosMultilaneMode_0 := 937, txt_DbVar_C0_RamRailWorkSafetyC0_WrongBasketPosMultilaneMode_0 := 938, txt_DbVar_C0_RamRailWorkSafetyC0_WrongTurretPosALOMode_0 := 939, txt_DbVar_C0_RamRailWorkSafetyC0_WrongPosition_0 := 940, txt_DbVar_C0_RamRailWorkSafetyC0_ReduceSpeedRotTurretClockwise_0 := 941, txt_DbVar_C0_RamRailWorkSafetyC0_ReduceSpeedRotTurretCounterClock_0 := 942, txt_DbVar_C0_RamRailWorkSafetyC0_ReduceSpeedArrowArmDown_0 := 943, txt_DbVar_C0_RamRailWorkSafetyC0_StopRotTurretClockwise_0 := 944, txt_DbVar_C0_RamRailWorkSafetyC0_StopRotTurretCounterClockwise_0 := 945, txt_DbVar_C0_RamRailWorkSafetyC0_StopRotBasketClockwise_0 := 946, txt_DbVar_C0_RamRailWorkSafetyC0_StopRotBasketCounterClockwise_0 := 947, txt_DbVar_C0_RamRailWorkSafetyC0_StopArrowArmDown_0 := 948, txt_DbVar_C0_RamRailWorkSafetyC0_StopTelescopeOut_0 := 949, txt_DbVar_C0_RamRailWorkSafetyC0_TurretInRearZone_0 := 950, txt_DbVar_C0_RamRailWorkSafetyC0_TurretInFrontZone_0 := 951, txt_DbVar_C0_RamRailWorkSafetyC0_ArrowArmInLowerZone_0 := 952, txt_DbVar_C0_RamRailWorkSafetyC0_TestFranceConfig_0 := 953, txt_DbVar_C0_RamRailWorkSafetyC0_TestAbutementBasketTrackSide_0 := 954, txt_DbVar_C0_RamRailWorkSafetyC0_TestAbutementBasketCenteredSide_0 := 955, txt_DbVar_C0_RamRailWorkSafetyC0_TestBasketLeftSideSensor_0 := 956, txt_DbVar_C0_RamRailWorkSafetyC0_TestBasketRightSideSensor_0 := 957, txt_DbVar_C0_RamRailWorkSafetyC0_TestTelescopInSensor_0 := 958, txt_DbVar_C0_RamRailWorkSafetyC0_TestTurretAngularPosition_0 := 959, txt_DbVar_C0_RamRailWorkSafetyC0_TestArrowArmAngularPosition_0 := 960, txt_DbVar_C0_RamRailWorkSafetyC0_AbutmentWorkMode_0 := 961, txt_DbVar_C0_RamTransportPosC0_DeltaOffRailTransportZone_0 := 962, txt_DbVar_C0_RamTransportPosC0_ArrowOffRailTransportZone_0 := 963, txt_DbVar_C0_RamTransportPosC0_TransportPosition_0 := 964, txt_DbVar_C0_NvParamTransportPosC0_DeltaArmTres_0 := 965, txt_DbVar_C0_NvParamTransportPosC0_DeltaArmHyst_0 := 966, txt_DbVar_C0_NvParamTransportPosC0_ArrowArmThres_0 := 967, txt_DbVar_C0_NvParamTransportPosC0_ArrowArmHyst_0 := 968, txt_DbVar_C0_NvParamTransportPosC0_TurretAngleThres_0 := 969, txt_DbVar_C0_RamBreakInBrakeC0_BreakInBrakeOffRailMode_0 := 970, txt_DbVar_C0_RamBreakInBrakeC0_ForceOsciServiceBrake_0 := 971, txt_DbVar_C0_RamBreakInBrakeC0_ForceFixeServiceBrake_0 := 972, txt_DbVar_C0_RamBreakInBrakeC0_ForceOsciParkBrake_0 := 973, txt_DbVar_C0_RamBreakInBrakeC0_ForceFixeParkBrake_0 := 974, txt_DbVar_C0_RamBreakInBrakeC0_StopMovementByBreakInBrake_0 := 975, txt_DbVar_C0_RamBreakInBrakeC0_IncoherencePosAxleAndTestMode_0 := 976, txt_DbVar_C0_RamBreakInBrakeC0_AdvancementPeriod_0 := 977, txt_DbVar_C0_RamBreakInBrakeC0_BreakInBrakeRunning_0 := 978, txt_DbVar_C0_RamBreakInBrakeC0_SimuOsciServiceBrakeSelect_0 := 979, txt_DbVar_C0_RamBreakInBrakeC0_SimuFixeServiceBrakeSelect_0 := 980, txt_DbVar_C0_RamBreakInBrakeC0_Simu2ServiceBrakesSelect_0 := 981, txt_DbVar_C0_RamBreakInBrakeC0_AuthorizeTransRailByBreakInBrake_0 := 982, txt_DbVar_C0_RamBreakInBrakeC0_ServiceBrakeSelected_0 := 983, txt_DbVar_C0_RamBreakInBrakeC0_AdvancementPeriodMs10_0 := 984, txt_DbVar_C0_RamBreakInBrakeC0_OsciServiceBrakinBrakeOn_0 := 985, txt_DbVar_C0_RamBreakInBrakeC0_FixeServiceBrakinBrakeOn_0 := 986, txt_DbVar_C0_RamBreakInBrakeC0_BothServiceBrakinBrakeOn_0 := 987, txt_DbVar_C0_RamSelectControlPost_SelectedControlPost_0 := 988, txt_DbVar_C0_RamSelectControlPost_EnableBuzzer_0 := 989, txt_DbVar_C0_RamSelectControlPost_SlopeIsLow_0 := 990, txt_DbVar_C0_RamSelectControlPost_SlopeIsHigh_0 := 991, txt_DbVar_C0_RamSelectControlPost_AllNacelleCommandsDisabled_0 := 992, txt_DbVar_C0_RamSelectControlPost_AllRadioCommandsDisabled_0 := 993, txt_DbVar_C0_RamSelectControlPost_AllTurretCommandsDisabled_0 := 994, txt_DbVar_C0_RamSelectControlPost_SimuSlope_0 := 995, txt_DbVar_C0_RamSelectControlPost_AllConsigneAdvancementDisabled_0 := 996, txt_DbVar_C0_RamSelectControlPost_AuthorizedRadioElementsPosition_0 := 997, txt_DbVar_C0_NvParamSelectControlPost_SlopeLowThresAbs_0 := 998, txt_DbVar_C0_NvParamSelectControlPost_SlopeLowHystRel_0 := 999, txt_DbVar_C0_NvParamSelectControlPost_SlopeHighThresAbs_0 := 1000, txt_DbVar_C0_NvParamSelectControlPost_SlopeHighHystRel_0 := 1001, txt_DbVar_C0_NvParamSelectControlPost_SlopeCrawlerMaxTres_0 := 1002, txt_DbVar_C0_RamEvision4C0_LifeByte_0 := 1003, txt_DbVar_C0_RamEvision4C0_gDelta_Arm_Move_Up_0 := 1004, txt_DbVar_C0_RamEvision4C0_gDelta_Arm_Move_Down_0 := 1005, txt_DbVar_C0_RamEvision4C0_gArrow_Move_Up_0 := 1006, txt_DbVar_C0_RamEvision4C0_gArrow_Move_Down_0 := 1007, txt_DbVar_C0_RamEvision4C0_gPendular_Move_Up_0 := 1008, txt_DbVar_C0_RamEvision4C0_gPendular_Move_Down_0 := 1009, txt_DbVar_C0_RamEvision4C0_gTelescope_Move_Out_0 := 1010, txt_DbVar_C0_RamEvision4C0_gTelescope_Move_In_0 := 1011, txt_DbVar_C0_RamEvision4C0_gBasket_Inclinaison_Move_Up_0 := 1012, txt_DbVar_C0_RamEvision4C0_gBasket_Inclinaison_Move_Down_0 := 1013, txt_DbVar_C0_RamEvision4C0_gTurret_Rotate_ClockWise_0 := 1014, txt_DbVar_C0_RamEvision4C0_gTurret_Rotate_Counter_ClockWise_0 := 1015, txt_DbVar_C0_RamEvision4C0_gBasket_Rotate_ClockWise_0 := 1016, txt_DbVar_C0_RamEvision4C0_gBasket_Rotate_Counter_ClockWise_0 := 1017, txt_DbVar_C0_RamEvision4C0_gKeyRpmSelect_0 := 1018, txt_DbVar_C0_RamEvision4C0_gKeyRpmOff_0 := 1019, txt_DbVar_C0_RamEvision4C0_gForcingWhiteRaillight_0 := 1020, txt_DbVar_C0_RamEvision4C0_gForcingNeons_0 := 1021, txt_DbVar_C0_RamEvision4C0_gKeyCalibMin_0 := 1022, txt_DbVar_C0_RamEvision4C0_gKeyCalibMax_0 := 1023, txt_DbVar_C0_RamEvision4C0_gKeyCalibValid_0 := 1024, txt_DbVar_C0_RamEvision4C0_gElementChoice_0 := 1025, txt_DbVar_C0_RamEvision4C0_gKeyCalibMax2_0 := 1026, txt_DbVar_C0_RamEvision4C0_gKeySlopeLgReset_0 := 1027, txt_DbVar_C0_RamEvision4C0_gKeySlopeTrReset_0 := 1028, txt_DbVar_C0_NvParamAlarmC0_TempTrackOverFaultThres_0 := 1029, txt_DbVar_C0_NvParamAlarmC0_TempRailOverFaultThres_0 := 1030, txt_DbVar_C0_NvParamAlarmC0_TempTrackOverAlarmThres_0 := 1031, txt_DbVar_C0_NvParamAlarmC0_TempRailOverAlarmThres_0 := 1032, txt_DbVar_C0_NvParamAlarmC0_SpeedSensorsToleranceThres_0 := 1033, txt_DbVar_C0_NvParamAlarmC0_SlopeLongToleranceThres_0 := 1034, txt_DbVar_C0_NvParamAlarmC0_BlockOscillationAxlePressure_0 := 1035, txt_DbVar_C0_NvParamAlarmC0_UnblockOscillationAxlePressure_0 := 1036, txt_DbVar_C0_NvParamAlarmC0_MinServiceBrakeFaultPressure_0 := 1037, txt_DbVar_C0_NvParamAlarmC0_MaxServiceBrakeFaultPressure_0 := 1038, txt_DbVar_C0_NvParamAlarmC0_SlopeTransToleranceThres_0 := 1039, txt_DbVar_C0_NvParamAlarmC0_MinTransPressureWithoutHook_0 := 1040, txt_DbVar_C0_NvParamAlarmC0_TurretSensorToleranceThres_0 := 1041, txt_DbVar_C0_NvParamAlarmC0_MinAlarmJoyDeltaArmPrctBat_0 := 1042, txt_DbVar_C0_NvParamAlarmC0_MaxAlarmJoyDeltaArmPrctBat_0 := 1043, txt_DbVar_C0_NvParamAlarmC0_MinAlarmJoyArrowArmPrctBat_0 := 1044, txt_DbVar_C0_NvParamAlarmC0_MaxAlarmJoyArrowArmPrctBat_0 := 1045, txt_DbVar_C0_NvParamAlarmC0_MinAlarmJoyTelescopeArmPrctBat_0 := 1046, txt_DbVar_C0_NvParamAlarmC0_MaxAlarmJoyTelescopeArmPrctBat_0 := 1047, txt_DbVar_C0_NvParamAlarmC0_MinAlarmJoyRotTurretArmPrctBat_0 := 1048, txt_DbVar_C0_NvParamAlarmC0_MaxAlarmJoyRotTurretArmPrctBat_0 := 1049, txt_DbVar_C0_NvParamAlarmC0_MinAlarmJoyAdvancementPrctBat_0 := 1050, txt_DbVar_C0_NvParamAlarmC0_MaxAlarmJoyAdvancementPrctBat_0 := 1051, txt_DbVar_C0_NvParamAlarmC0_HystTempTrans_0 := 1052, txt_DbVar_C0_NvParamAlarmC0_ReduceTrackSpeedPercent_0 := 1053, txt_DbVar_C0_NvParamAlarmC0_CptPressureBrakeFaultMax_0 := 1054, txt_DbVar_C0_NvParamAlarmC0_BypassAlarmActiveC0_0 := 1055, txt_DbVar_C0_NvParamAlarmC0_TimeBypassFault_0 := 1056, txt_DbVar_C0_NvParamAlarmC0_AU_THER_PRESSION_DEF_TRANS_0 := 1057, txt_DbVar_C0_NvParamAlarmC0_AU_ELEC_PRESSION_DEF_DMC_0 := 1058, txt_DbVar_C0_NvParamAlarmC0_cptTimeDetectPumpTransMax_0 := 1059, txt_DbVar_C0_NvParamAlarmC0_cptTimeDetectPvgTransMax_0 := 1060, txt_DbVar_C0_RamEcuAlarmC0_RamEcuAlarmC0_1_0 := 1061, txt_DbVar_C0_RamEcuAlarmC0_FaultPumpTrans_0 := 1062, txt_DbVar_C0_RamEcuAlarmC0_TimeDetectPumpTrans_0 := 1063, txt_DbVar_C0_RamEcuAlarmC0_MemFaultThermicPumpTrans_0 := 1064, txt_DbVar_C0_RamEcuAlarmC0_FaultPvgTransElectric_0 := 1065, txt_DbVar_C0_RamEcuAlarmC0_TimeDetectPvgTrans_0 := 1066, txt_DbVar_C0_RamEcuAlarmC0_MemFaultDMCTransElectric_0 := 1067, txt_DbVar_C0_RamEcuAlarmC0_FaultThermicPumpOrElecticDmc_0 := 1068, txt_DbVar_C0_RamEcuC0RcvFailluresFromC1_Dm_Inc_Pos_Folded_Delta_Arrow_0 := 1069, txt_DbVar_C0_RamEcuC0RcvFailluresFromC1_Dm_Active_Help_0 := 1070, txt_DbVar_C0_RamEcuC0RcvFailluresFromC1_Dm_Ev_Bypass_Fault_0 := 1071, txt_DbVar_C0_RamEcuC0RcvFailluresFromC1_OutOfRangeTransmissionPressure_0 := 1072, txt_DbVar_C0_RamEcuC0RcvFailluresFromC1_Dm_Overload_Detected_By_C1_0 := 1073, txt_DbVar_C0_RamMastDisplayMeasureC0_ErrorCodeInit_0 := 1074, txt_DbVar_C0_RamMastDisplayMeasureC0_ErrorCodeWrite_0 := 1075, txt_DbVar_C0_RamMastDisplayMeasureC0_RetDataBytesSent_0 := 1076, txt_DbVar_C0_RamMastDisplayMeasureC0_DisplayedDigit1_0 := 1077, txt_DbVar_C0_RamMastDisplayMeasureC0_DisplayedDigit2_0 := 1078, txt_DbVar_C0_RamMastDisplayMeasureC0_DisplayedDigit3_0 := 1079, txt_DbVar_C0_RamMastDisplayMeasureC0_DisplayedDigit4_0 := 1080, txt_DbVarArrDescr_C0_RamMastDisplayMeasureC0_SentDataArray := 1081, txt_DbVar_C0_RamMastDisplayMeasureC0_SentDataArray_0 := 1082, txt_DbVar_C0_RamMastDisplayMeasureC0_SentDataArray_1 := 1083, txt_DbVar_C0_RamMastDisplayMeasureC0_SentDataArray_2 := 1084, txt_DbVar_C0_RamMastDisplayMeasureC0_SentDataArray_3 := 1085, txt_DbVar_C0_RamMastDisplayMeasureC0_SentDataArray_4 := 1086, txt_DbVar_C0_RamMastDisplayMeasureC0_SentDataArray_5 := 1087, txt_DbVar_C0_RamMastDisplayMeasureC0_SentDataArray_6 := 1088, txt_DbVar_C0_RamMastDisplayMeasureC0_SentDataArray_7 := 1089, txt_DbVar_C0_NvParamMastDisplayC0_MastDisplayRefreshCycleTime_0 := 1090, txt_DbVar_C0_RamData4C0RcvFromC1_NoMovementRunning_0 := 1091, txt_DbVar_C0_RamData4C0RcvFromC1_StopMoveLimitEnvelop_0 := 1092, txt_DbVar_C0_RamData4C0RcvFromC1_TransmissionPressureFault_0 := 1093, txt_DbVar_C0_RamData4C0RcvFromC1_LynxOnAllMvts_0 := 1094, txt_DbVar_C0_RamData4C0RcvFromC1_Signal_4_0 := 1095, txt_DbVar_C0_RamData4C0RcvFromC1_Signal_5_0 := 1096, txt_DbVar_C0_RamData4C0RcvFromC1_Signal_6_0 := 1097, txt_DbVar_C0_RamData4C0RcvFromC1_Signal_7_0 := 1098, txt_DbVar_C0_RamData4C0RcvFromC1_Signal_8_0 := 1099, txt_DbVar_C0_RamData4C0RcvFromC1_BypassPressureSensorValue_0 := 1100, txt_DbVar_C0_RamData4C0RcvFromC1_Signal_10_0 := 1101, txt_DbVar_C0_RamData4C0RcvFromC1_Signal_11_0 := 1102, txt_DbVar_C0_RamData4C0RcvFromC1_PerformAutoriseTransArrow_0 := 1103, txt_DbVar_C0_RamData4C0RcvFromC1_ValidTelescopeSectorSlope_0 := 1104, txt_DbVar_C0_RamData4C0RcvFromC1_ValidTelescopeFirstSectorSlope_0 := 1105, txt_DbVar_C0_RamData4C0RcvFromC1_PostInterdictionMastSNCF_0 := 1106, txt_DbVar_C0_RamData4C0RcvFromC1_InterdictOfNacelTurretPost_0 := 1107, txt_DbVar_C0_RamData4C0RcvFromC1_MastPanthoFoldedSNCF_0 := 1108, txt_DbVar_C0_NvParamGreenEffC0_MaxPvgTransRailElectricAv_0 := 1109, txt_DbVar_C0_NvParamGreenEffC0_MaxPvgTransRailElectricAr_0 := 1110, txt_DbVar_C0_NvParamGreenEffC0_MinPvgTransRailElectricAv_0 := 1111, txt_DbVar_C0_NvParamGreenEffC0_MinPvgTransRailElectricAr_0 := 1112, txt_DbVar_C0_NvParamGreenEffC0_TransRailElectricRampTimeAcc_0 := 1113, txt_DbVar_C0_NvParamGreenEffC0_TransRailElectricRampTimeDec_0 := 1114, txt_DbVar_C0_NvParamGreenEffC0_TransRailElectricRampTimeStop_0 := 1115, txt_DbVar_C0_NvParamGreenEffC0_ElectricPumpPressureMax_0 := 1116, txt_DbVar_C0_NvParamGreenEffC0_ElectricPumpPressureHyst_0 := 1117, txt_DbVar_C0_NvParamGreenEffC0_ELECTRIC_MOTOR_RPM_TRANS_MAX_0 := 1118, txt_DbVar_C0_NvParamGreenEffC0_ELECTRIC_MOTOR_RPM_TRANS_MIN_0 := 1119, txt_DbVar_C0_NvParamGreenEffC0_MIN_PVG_TRANS_HIGH_50_0 := 1120, txt_DbVar_C0_NvParamGreenEffC0_MIN_PVG_TRANS_LOW_50_0 := 1121, txt_DbVar_C0_NvParamGreenEffC0_RAMP_TIME_REGEN_THERMIC_0 := 1122, txt_DbVar_C0_NvParamGreenEffC0_RegenPumpPressureMax_0 := 1123, txt_DbVar_C0_NvParamGreenEffC0_RegenPumpPressureReset_0 := 1124, txt_DbVar_C0_NvParamGreenEffC0_CURRENT_RESET_REGEN_THERMIC_0 := 1125, txt_DbVar_C0_NvParamGreenEffC0_CURRENT_MIN_REGEN_THERMIC_0 := 1126, txt_DbVar_C0_NvParamGreenEffC0_CURRENT_MAX_REGEN_THERMIC_0 := 1127, txt_DbVar_C0_NvParamGreenEffC0_CURRENT_DRIVE_LIMIT_ELECTRIC_0 := 1128, txt_DbVar_C0_NvParamGreenEffC0_BATTERY_LOW_LEVEL_SOC_0 := 1129, txt_DbVar_C0_NvParamGreenEffC0_MinVoltageDcConverter_0 := 1130, txt_DbVar_C0_NvParamGreenEffC0_NbrCycleFaultDcConverter_0 := 1131, txt_DbVar_C0_NvParamGreenEffC0_REGEN_BRAKE_RPM_MODE_AUTO_0 := 1132, txt_DbVar_C0_NvParamGreenEffC0_REGEN_BRAKE_TORQUE_MODE_AUTO_0 := 1133, txt_DbVar_C0_NvParamGreenEffC0_REGEN_BRAKE_RPM_MODE_HIGH_0 := 1134, txt_DbVar_C0_NvParamGreenEffC0_REGEN_BRAKE_TORQUE_MODE_HIGH_0 := 1135, txt_DbVar_C0_NvParamGreenEffC0_NbrSamplesAverageRpm_0 := 1136, txt_DbVar_C0_NvParamGreenEffC0_RegenPumpPressureHyst_0 := 1137, txt_DbVar_C0_NvParamGreenEffC0_RegenBrakeTorqueFromPressurCoefK_0 := 1138, txt_DbVar_C0_NvParamGreenEffC0_RegenBrakeTorqueFromPressurRange_0 := 1139, txt_DbVar_C0_RamGreenEffC0_AutorizeTransRailElectric_0 := 1140, txt_DbVar_C0_RamGreenEffC0_PvgTransRailElectricConsigne_0 := 1141, txt_DbVar_C0_RamGreenEffC0_ElectricPumpPressureExceeded_0 := 1142, txt_DbVar_C0_RamGreenEffC0_StopRampPvgTransRailElectric_0 := 1143, txt_DbVar_C0_RamGreenEffC0_TransRailElectricRampOngoing_0 := 1144, txt_DbVar_C0_RamGreenEffC0_TransRailThermiqueRampOngoing_0 := 1145, txt_DbVar_C0_RamGreenEffC0_RpmPvgTransRail_0 := 1146, txt_DbVar_C0_RamGreenEffC0_PictoReloadBatteryImpossible_0 := 1147, txt_DbVar_C0_RamGreenEffC0_BatteryLowLevel_0 := 1148, txt_DbVar_C0_RamGreenEffC0_ElectricPumpPressureMaxRegen_0 := 1149, txt_DbVar_C0_RamGreenEffC0_ElectricPumpPressureResetRegen_0 := 1150, txt_DbVar_C0_RamGreenEffC0_AutorizeRazController_0 := 1151, txt_DbVar_C0_RamGreenEffC0_VoltageDcConverterFault_0 := 1152, txt_DbVar_C0_RamGreenEffC0_BattErrorCode1_0 := 1153, txt_DbVar_C0_RamGreenEffC0_PictoAskResartController_0 := 1154, txt_DbVar_C0_RamFlashBatteryC0_Ibatt_ist_0 := 1155, txt_DbVar_C0_RamFlashBatteryC0_Vbatt_ist_0 := 1156, txt_DbVar_C0_RamFlashBatteryC0_Batt_Soc_0 := 1157, txt_DbVar_C0_RamFlashBatteryC0_Batt_PowerReductionRatio_0 := 1158, txt_DbVar_C0_RamFlashBatteryC0_Batt_RecoveryReductionRatio_0 := 1159, txt_DbVar_C0_RamFlashBatteryC0_Batt_ErrorCode1_0 := 1160, txt_DbVar_C0_RamFlashBatteryC0_Batt_ErrorValue1_0 := 1161, txt_DbVar_C0_RamFlashBatteryC0_Batt_RegenAuthorized_0 := 1162, txt_DbVar_C0_RamDMC_C0_DC_RpmRequest_0 := 1163, txt_DbVar_C0_RamDMC_C0_DC_AI2_StaticBrakeTorqueLimit_0 := 1164, txt_DbVar_C0_RamDMC_C0_DC_GeneratorRegenBattCurLimit_0 := 1165, txt_DbVar_C0_RamDMC_C0_DC_ForwardByte6Bit0_0 := 1166, txt_DbVar_C0_RamDMC_C0_DC_BackwardByte6Bit1_0 := 1167, txt_DbVar_C0_RamDMC_C0_DC_FootSwitchByte6Bit2_0 := 1168, txt_DbVar_C0_RamDMC_C0_DC_InterlockByt6Bit3_0 := 1169, txt_DbVar_C0_RamDMC_C0_DC_RegenEnableByte6Bit6_0 := 1170, txt_DbVar_C0_RamDMC_C0_DC_RollOverCount_0 := 1171, txt_DbVar_C0_RamDMC_C0_BCL_HMI_DriveBattCurLimit_0 := 1172, txt_DbVar_C0_RamDMC_C0_BCL_HMI_RegenBattCurLimit_0 := 1173, txt_DbVar_C0_RamDMC_C0_BCL_HMI_BattSOC_0 := 1174, txt_DbVar_C0_RamDMC_C0_BCL_RollOverCount_0 := 1175, txt_DbVar_C0_RamDMC_C0_MS_ActualSpeedRpm_0 := 1176, txt_DbVar_C0_RamDMC_C0_MS_BattCur_0 := 1177, txt_DbVar_C0_RamDMC_C0_MS_RollOverCount_0 := 1178, txt_DbVar_C0_RamDMC_C0_MS_FaultCode_0 := 1179, txt_DbVar_C0_RamDMC_C0_MS_FaultSubCode_0 := 1180, txt_DbVar_C0_RamDMC_C0_DS_MotorCur_0 := 1181, txt_DbVar_C0_RamDMC_C0_DS_DriveStatusIndicator_0 := 1182, txt_DbVar_C0_RamDMC_C0_DS_SpeedLimitIndicator_0 := 1183, txt_DbVar_C0_RamDMC_C0_DS_ActualTorque_0 := 1184, txt_DbVar_C0_RamDMC_C0_DS_TorqueLimitIndicator_0 := 1185, txt_DbVar_C0_RamDMC_C0_DS_RollOverCount_0 := 1186, txt_DbVar_C0_RamDMC_C0_CS_ControlerTemp_0 := 1187, txt_DbVar_C0_RamDMC_C0_CS_MotorTemp_0 := 1188, txt_DbVar_C0_RamDMC_C0_CS_MotorLimitIndicator_0 := 1189, txt_DbVar_C0_RamDMC_C0_CS_RollOverCount_0 := 1190, txt_DbVar_C0_RamDMC_C0_CS_BattVoltage_0 := 1191, txt_DbVar_C0_RamDMC_C0_CS_BattDischargeIndicatorValue_0 := 1192, txt_DbVar_C0_RamDMC_C0_WaitingHeartbeat_0 := 1193, txt_DbVar_C0_RamDMC_C0_TimeOutDmcHeartbeat_0 := 1194, txt_DbVar_C0_RamDMC_C0_DmcHeartbeat_0 := 1195, txt_DbVar_C0_RamDMC_C0_PowerOnOkDmc_0 := 1196, txt_DbVar_C0_RamDMC_C0_OperationnalDmc_0 := 1197, txt_DbVar_C0_RamDMC_C0_GoToOperationnal_0 := 1198, txt_DbVar_C0_RamDMC_C0_NewGoToOperationnal_0 := 1199, txt_DbVar_C0_RamDMC_C0_SendCommandNMT_0 := 1200, txt_DbVar_C0_RamDMC_C0_StepRazDmc_0 := 1201, txt_DbVar_C0_RamDMC_C0_CommandRazDmcOnGoing_0 := 1202, txt_DbVar_C0_RamDMC_C0_Dig4InputCommandSTO_0 := 1203, txt_DbVar_C0_RamDMC_C0_ActiveFaultRazDmc_0 := 1204, txt_DbVar_C0_RamDMC_C0_ActiveFaultDmc_0 := 1205, txt_DbVar_C1_RamEcuInputsC1_DeltaArmAngularSensorState_0 := 1206, txt_DbVar_C1_RamEcuInputsC1_DeltaArmAngularSensorValue_0 := 1207, txt_DbVar_C1_RamEcuInputsC1_DeltaArmAngleValue_0 := 1208, txt_DbVar_C1_RamEcuInputsC1_DeltaArmAngularSensorRawValueMas_0 := 1209, txt_DbVar_C1_RamEcuInputsC1_DeltaArmAngularSensorRawValueSla_0 := 1210, txt_DbVar_C1_RamEcuInputsC1_ArrowArmAngularSensorState_0 := 1211, txt_DbVar_C1_RamEcuInputsC1_ArrowArmAngularSensorValue_0 := 1212, txt_DbVar_C1_RamEcuInputsC1_ArrowArmAngleValue_0 := 1213, txt_DbVar_C1_RamEcuInputsC1_ArrowArmAngularSensorRawValueMas_0 := 1214, txt_DbVar_C1_RamEcuInputsC1_ArrowArmAngularSensorRawValueSla_0 := 1215, txt_DbVar_C1_RamEcuInputsC1_GasGaugeValue_0 := 1216, txt_DbVar_C1_RamEcuInputsC1_GasGaugeRawValue_0 := 1217, txt_DbVar_C1_RamEcuInputsC1_Aru1State_0 := 1218, txt_DbVar_C1_RamEcuInputsC1_Aru1RawValue_0 := 1219, txt_DbVar_C1_RamEcuInputsC1_Aru2State_0 := 1220, txt_DbVar_C1_RamEcuInputsC1_Aru2RawValue_0 := 1221, txt_DbVar_C1_RamEcuInputsC1_EntryTelescopeFdcSensorState_0 := 1222, txt_DbVar_C1_RamEcuInputsC1_EntryTelescopeFdcSensorRawValue_0 := 1223, txt_DbVar_C1_RamEcuInputsC1_FoldedDeltaArmSensorState_0 := 1224, txt_DbVar_C1_RamEcuInputsC1_FoldedDeltaArmSensorRawValue_0 := 1225, txt_DbVar_C1_RamEcuInputsC1_FoldedBoomArmSensorState_0 := 1226, txt_DbVar_C1_RamEcuInputsC1_FoldedBoomArmSensorRawValue_0 := 1227, txt_DbVar_C1_RamEcuInputsC1_ForcingMotorRegimeState_0 := 1228, txt_DbVar_C1_RamEcuInputsC1_ForcingMotorRegimeRawValue_0 := 1229, txt_DbVar_C1_RamEcuInputsC1_ActiveHelpState_0 := 1230, txt_DbVar_C1_RamEcuInputsC1_ActiveHelpRawValue_0 := 1231, txt_DbVar_C1_RamEcuInputsC1_OilPressureState_0 := 1232, txt_DbVar_C1_RamEcuInputsC1_OilPressureRawValue_0 := 1233, txt_DbVar_C1_RamEcuInputsC1_WaterTemperatureState_0 := 1234, txt_DbVar_C1_RamEcuInputsC1_WaterTemperatureRawValue_0 := 1235, txt_DbVar_C1_RamEcuInputsC1_StopMotorInfoState_0 := 1236, txt_DbVar_C1_RamEcuInputsC1_StopMotorInfoRawValue_0 := 1237, txt_DbVar_C1_RamEcuInputsC1_TurretPostSelectorState_0 := 1238, txt_DbVar_C1_RamEcuInputsC1_TurretPostSelectorRawValue_0 := 1239, txt_DbVar_C1_RamEcuInputsC1_RadioPostSelectorState_0 := 1240, txt_DbVar_C1_RamEcuInputsC1_RadioPostSelectorRawValue_0 := 1241, txt_DbVar_C1_RamEcuInputsC1_NacellePostSelectorState_0 := 1242, txt_DbVar_C1_RamEcuInputsC1_NacellePostSelectorRawValue_0 := 1243, txt_DbVar_C1_RamEcuInputsC1_RegimeMotorAlternatorRpm_0 := 1244, txt_DbVar_C1_RamEcuInputsC1_AlternatorChargeOkState_0 := 1245, txt_DbVar_C1_RamEcuInputsC1_AlternatorChargeOkValue_0 := 1246, txt_DbVar_C1_RamEcuInputsC1_Transmission1PressureSensorState_0 := 1247, txt_DbVar_C1_RamEcuInputsC1_Transmission1PressureSensorValue_0 := 1248, txt_DbVar_C1_RamEcuInputsC1_Transmission2PressureSensorState_0 := 1249, txt_DbVar_C1_RamEcuInputsC1_Transmission2PressureSensorValue_0 := 1250, txt_DbVar_C1_RamEcuInputsC1_FaultPvgDeltaArmState_0 := 1251, txt_DbVar_C1_RamEcuInputsC1_FaultPvgDeltaArmRawValue_0 := 1252, txt_DbVar_C1_RamEcuInputsC1_FaultPvgArrowArmState_0 := 1253, txt_DbVar_C1_RamEcuInputsC1_FaultPvgArrowArmRawValue_0 := 1254, txt_DbVar_C1_RamEcuInputsC1_FaultPvgTelescopeArmState_0 := 1255, txt_DbVar_C1_RamEcuInputsC1_FaultPvgTelescopeArmRawValue_0 := 1256, txt_DbVar_C1_RamEcuInputsC1_FaultPvgEvProTorState_0 := 1257, txt_DbVar_C1_RamEcuInputsC1_FaultPvgEvProTorRawValue_0 := 1258, txt_DbVar_C1_RamEcuInputsC1_BypassPressureSensorState_0 := 1259, txt_DbVar_C1_RamEcuInputsC1_BypassPressureSensorValue_0 := 1260, txt_DbVar_C1_RamEcuInputsC1_BypassPressureSensorRawValue_0 := 1261, txt_DbVar_C1_RamEcuInputsC1_StarterMotorState_0 := 1262, txt_DbVar_C1_RamEcuInputsC1_StarterMotorRawValue_0 := 1263, txt_DbVar_C1_RamEcuInputsC1_OilTankTemperatureState_0 := 1264, txt_DbVar_C1_RamEcuInputsC1_OilTankTemperatureValue_0 := 1265, txt_DbVar_C1_RamEcuInputsC1_OilTankTemperatureRawValue_0 := 1266, txt_DbVar_C1_RamEcuOutputsC1_BlueFireCommand_0 := 1267, txt_DbVar_C1_RamEcuOutputsC1_BlueFireValue_0 := 1268, txt_DbVar_C1_RamEcuOutputsC1_OrangeFlashingLightCommand_0 := 1269, txt_DbVar_C1_RamEcuOutputsC1_OrangeFlashingLightValue_0 := 1270, txt_DbVar_C1_RamEcuOutputsC1_AntiStartupCommand_0 := 1271, txt_DbVar_C1_RamEcuOutputsC1_AntiStartupValue_0 := 1272, txt_DbVar_C1_RamEcuOutputsC1_StopMotorCommand_0 := 1273, txt_DbVar_C1_RamEcuOutputsC1_WarmingCommand_0 := 1274, txt_DbVar_C1_RamEcuOutputsC1_EvBypassCommand_0 := 1275, txt_DbVar_C1_RamEcuOutputsC1_EvBypassValue_0 := 1276, txt_DbVar_C1_RamEcuOutputsC1_SupplyPvgDeltaArmCommand_0 := 1277, txt_DbVar_C1_RamEcuOutputsC1_SupplyPvgDeltaArmValue_0 := 1278, txt_DbVar_C1_RamEcuOutputsC1_SupplyPvgArrowArmCommand_0 := 1279, txt_DbVar_C1_RamEcuOutputsC1_SupplyPvgArrowArmValue_0 := 1280, txt_DbVar_C1_RamEcuOutputsC1_SupplyPvgTelescopeArmCommand_0 := 1281, txt_DbVar_C1_RamEcuOutputsC1_SupplyPvgTelescopeArmValue_0 := 1282, txt_DbVar_C1_RamEcuOutputsC1_SupplyPvgPropEvTorCommand_0 := 1283, txt_DbVar_C1_RamEcuOutputsC1_SupplyPvgPropEvTorValue_0 := 1284, txt_DbVar_C1_RamEcuOutputsC1_EvPropMotorAcceleratorCommand_0 := 1285, txt_DbVar_C1_RamEcuOutputsC1_EvPropGeneratorState_0 := 1286, txt_DbVar_C1_RamEcuOutputsC1_EvPropGeneratorCommand_0 := 1287, txt_DbVar_C1_RamEcuOutputsC1_EvPropGeneratorCurrent_0 := 1288, txt_DbVar_C1_RamEcuOutputsC1_NoisemakerState_0 := 1289, txt_DbVar_C1_RamEcuOutputsC1_NoisemakerCommand_0 := 1290, txt_DbVar_C1_RamEcuOutputsC1_EvRotationTurretCtClockwiseState_0 := 1291, txt_DbVar_C1_RamEcuOutputsC1_EvRotTurretCtClockwiseCmdBool_0 := 1292, txt_DbVar_C1_RamEcuOutputsC1_EvRotationTurretClockwiseState_0 := 1293, txt_DbVar_C1_RamEcuOutputsC1_EvRotTurretClockwiseCmdBool_0 := 1294, txt_DbVar_C1_RamEcuOutputsC1_EvRotationBasketCtClockwiseState_0 := 1295, txt_DbVar_C1_RamEcuOutputsC1_EvRotationBasketCtClkWiseCmdBool_0 := 1296, txt_DbVar_C1_RamEcuOutputsC1_EvRotationBasketClockwiseState_0 := 1297, txt_DbVar_C1_RamEcuOutputsC1_EvRotationBasketClkWiseCmdBool_0 := 1298, txt_DbVar_C1_RamEcuOutputsC1_EvUpPendularState_0 := 1299, txt_DbVar_C1_RamEcuOutputsC1_EvUpPendularCommandBool_0 := 1300, txt_DbVar_C1_RamEcuOutputsC1_EvDownPendularState_0 := 1301, txt_DbVar_C1_RamEcuOutputsC1_EvDownPendularCommandBool_0 := 1302, txt_DbVar_C1_RamEcuOutputsC1_EvUpInclinaisonBasketState_0 := 1303, txt_DbVar_C1_RamEcuOutputsC1_EvUpInclinaisonBasketCmdBool_0 := 1304, txt_DbVar_C1_RamEcuOutputsC1_EvDownInclinaisonBasketState_0 := 1305, txt_DbVar_C1_RamEcuOutputsC1_EvDownInclinaisonBasketCommand_0 := 1306, txt_DbVar_C1_RamEcuOutputsC1_EvDownInclinaisonBasketCmdBool_0 := 1307, txt_DbVar_C1_RamEcuOutputsC1_EvDownInclinaisonBasketCurrent_0 := 1308, txt_DbVar_C1_RamEcuOutputsC1_PvgDeltaArmCommand_0 := 1309, txt_DbVar_C1_RamEcuOutputsC1_PvgDeltaArmVoltage_0 := 1310, txt_DbVar_C1_RamEcuOutputsC1_PvgArrowArmCommand_0 := 1311, txt_DbVar_C1_RamEcuOutputsC1_PvgArrowArmVoltage_0 := 1312, txt_DbVar_C1_RamEcuOutputsC1_PvgTelescopeArmCommand_0 := 1313, txt_DbVar_C1_RamEcuOutputsC1_PvgTelescopeArmVoltage_0 := 1314, txt_DbVar_C1_RamEcuOutputsC1_OverloadSecurityCommand_0 := 1315, txt_DbVar_C1_RamEcuOutputsC1_OverloadSecurityValue_0 := 1316, txt_DbVar_C1_RamEcuOutputsC1_SupllyTorSensorsCommand_0 := 1317, txt_DbVar_C1_RamEcuOutputsC1_SupllyTorSensorsValue_0 := 1318, txt_DbVar_C1_RamEcuOutputsC1_SupllyAnaSensorsCommand_0 := 1319, txt_DbVar_C1_RamEcuOutputsC1_SupllyAnaSensorsValue_0 := 1320, txt_DbVar_C1_RamEcuOutputsC1_EvSyncRotationCommand_0 := 1321, txt_DbVar_C1_RamEcuOutputsC1_EvSyncRotationValue_0 := 1322, txt_DbVar_C1_RamEcuOutputsC1_PvgEvTorCommand_0 := 1323, txt_DbVar_C1_RamEcuOutputsC1_PvgEvTorVoltage_0 := 1324, txt_DbVar_C1_RamEcuOutputsC1_EvUpPendularActivation_0 := 1325, txt_DbVar_C1_RamEcuOutputsC1_EvDownPendularActivation_0 := 1326, txt_DbVar_C1_RamEcuOutputsC1_EvRotBasketCtClkWiseActivation_0 := 1327, txt_DbVar_C1_RamEcuOutputsC1_EvRotBasketClkWiseActivation_0 := 1328, txt_DbVar_C1_RamEcuOutputsC1_EvUpIncliBasketActivation_0 := 1329, txt_DbVar_C1_RamEcuOutputsC1_EvDownIncliBasketActivation_0 := 1330, txt_DbVar_C1_RamEcuOutputsC1_EvRotTurretClockwiseActivation_0 := 1331, txt_DbVar_C1_RamEcuOutputsC1_EvRotTurretCtClockwiseActivation_0 := 1332, txt_DbVar_C1_RamEcuOutputsC1_EvSelectorRotTurretValue_0 := 1333, txt_DbVar_C1_RamEcuOutputsC1_EvSelectorRotTurretCmd_0 := 1334, txt_DbVar_C1_RamEcuOutputsC1_ReturnLowSideEvProAccMotorCmd_0 := 1335, txt_DbVar_C1_RamEcuOutputsC1_ReturnLowSideEvProGeneratorCmd_0 := 1336, txt_DbVar_C1_RamEcuOutputsC1_ReturnLowSideEvProGeneratorValue_0 := 1337, txt_DbVar_C1_RamEcuOutputsC1_EvUpAxleOscillantActivation_0 := 1338, txt_DbVar_C1_RamEcuOutputsC1_EvDownAxleOscillantActivation_0 := 1339, txt_DbVar_C1_RamEcuOutputsC1_EvUpAxleOscillantCmd_0 := 1340, txt_DbVar_C1_RamEcuOutputsC1_EvDownAxleOscillantCmd_0 := 1341, txt_DbVar_C1_RamEcuOutputsC1_EvUpAxleFixeActivation_0 := 1342, txt_DbVar_C1_RamEcuOutputsC1_EvDownAxleFixeActivation_0 := 1343, txt_DbVar_C1_RamEcuOutputsC1_EvUpAxleFixeCmd_0 := 1344, txt_DbVar_C1_RamEcuOutputsC1_EvDownAxleFixeCmd_0 := 1345, txt_DbVar_C1_RamEcuOutputsC1_EvUpMastMeasureActivation_0 := 1346, txt_DbVar_C1_RamEcuOutputsC1_EvUpMastMeasureCmd_0 := 1347, txt_DbVar_C1_RamEcuOutputsC1_EvDownMastMeasureActivation_0 := 1348, txt_DbVar_C1_RamEcuOutputsC1_EvDownMastMeasureCmd_0 := 1349, txt_DbVar_C1_RamEcuOutputsC1_WhiteLightAv15746Value_0 := 1350, txt_DbVar_C1_RamEcuOutputsC1_WhiteLightAv15746Command_0 := 1351, txt_DbVar_C1_RamEcuOutputsC1_EvCrawlerOnlyValue_0 := 1352, txt_DbVar_C1_RamEcuOutputsC1_EvCrawlerOnlyCommand_0 := 1353, txt_DbVar_C1_RamEcuOutputsC1_RelayReloadWithGeneratorCmd_0 := 1354, txt_DbVar_C1_RamEcuOutputsC1_RelayReloadWithGeneratorState_0 := 1355, txt_DbVar_C1_RamEcuOutputsC1_EvDevMvtsCmd_0 := 1356, txt_DbVar_C1_RamEcuOutputsC1_EvDevMvtsState_0 := 1357, txt_DbVar_C1_RamEcuOutputsC1_EvBoostRegenCmd_0 := 1358, txt_DbVar_C1_RamEcuOutputsC1_EvBoostRegenState_0 := 1359, txt_DbVar_C1_RamGeneralC1_LifeByte_0 := 1360, txt_DbVar_C1_RamGeneralC1_WatchdogState_0 := 1361, txt_DbVar_C1_RamGeneralC1_EcuVoltage_0 := 1362, txt_DbVar_C1_RamGeneralC1_BypassArmDelta_0 := 1363, txt_DbVar_C1_RamGeneralC1_BypassArmArrow_0 := 1364, txt_DbVar_C1_RamGeneralC1_BypassArmTelescope_0 := 1365, txt_DbVar_C1_RamGeneralC1_TestEvision_0 := 1366, txt_DbVar_C1_RamGeneralC1_PvgTorConsigneCommand_0 := 1367, txt_DbVar_C1_RamGeneralC1_PvgEvTorTurretCmd_0 := 1368, txt_DbVar_C1_RamGeneralC1_EngineOn_0 := 1369, txt_DbVar_C1_RamGeneralC1_gMotorCmd_0 := 1370, txt_DbVar_C1_RamGeneralC1_CounterRisingEdge_0 := 1371, txt_DbVar_C1_RamGeneralC1_CounterFallingEdge_0 := 1372, txt_DbVar_C1_RamGeneralC1_LifeBitRotBasket_0 := 1373, txt_DbVar_C1_RamGeneralC1_TestElevationActivation_0 := 1374, txt_DbVar_C1_RamGeneralC1_RotTurretBool_0 := 1375, txt_DbVar_C1_RamGeneralC1_ScalingJoysTurret_0 := 1376, txt_DbVar_C1_RamGeneralC1_ScalingJoysDeltaArm_0 := 1377, txt_DbVar_C1_RamGeneralC1_PvgDeltaArmConsigne_0 := 1378, txt_DbVar_C1_RamGeneralC1_ScalingJoysArrowArm_0 := 1379, txt_DbVar_C1_RamGeneralC1_PvgArrowArmConsigne_0 := 1380, txt_DbVar_C1_RamGeneralC1_ScalingJoysTelescopeArm_0 := 1381, txt_DbVar_C1_RamGeneralC1_PvgTelescopeArmConsigne_0 := 1382, txt_DbVarArrDescr_C1_RamGeneralC1_PvgTorVoltageRangeValue := 1383, txt_DbVar_C1_RamGeneralC1_PvgTorVoltageRangeValue_0 := 1384, txt_DbVar_C1_RamGeneralC1_PvgTorVoltageRangeValue_1 := 1385, txt_DbVar_C1_RamGeneralC1_PvgTorVoltageRangeValue_2 := 1386, txt_DbVar_C1_RamGeneralC1_PvgTorVoltageRangeValue_3 := 1387, txt_DbVar_C1_RamGeneralC1_PvgTorVoltageRangeValue_4 := 1388, txt_DbVar_C1_RamGeneralC1_ActiveWorkEnvelopLimit_0 := 1389, txt_DbVar_C1_RamGeneralC1_PortillonLadderClose_0 := 1390, txt_DbVar_C1_RamGeneralC1_ActiveFailure_0 := 1391, txt_DbVar_C1_RamGeneralC1_StopAllMovementsNacellePost_0 := 1392, txt_DbVar_C1_RamGeneralC1_AverageTimeCycle_0 := 1393, txt_DbVar_C1_RamGeneralC1_MaxTimeCycle_0 := 1394, txt_DbVar_C1_RamGeneralC1_TestRefreshParamBlockCurrent_0 := 1395, txt_DbVar_C1_RamGeneralC1_LynxOnAllMvts_0 := 1396, txt_DbVar_C1_RamGeneralC1_ReturnValStart48XsFunc_0 := 1397, txt_DbVar_C1_RamGeneralC1_IndexVersion48Xs_0 := 1398, txt_DbVar_C1_RamGeneralC1_TestElectricalIO_0 := 1399, txt_DbVar_C1_RamGeneralC1_Major_48XS_0 := 1400, txt_DbVar_C1_RamGeneralC1_Minor_48XS_0 := 1401, txt_DbVar_C1_RamGeneralC1_Patch_48XS_0 := 1402, txt_DbVar_C1_RamGeneralC1_Custom_48XS_0 := 1403, txt_DbVar_C1_RamGeneralC1_RunningStable48XS_0 := 1404, txt_DbVar_C1_RamGeneralC1_BlinkLow_0 := 1405, txt_DbVar_C1_RamGeneralC1_FaultyValue_0 := 1406, txt_DbVar_C1_RamGeneralC1_DeviceNum_0 := 1407, txt_DbVar_C1_RamGeneralC1_ErrorCode_0 := 1408, txt_DbVar_C1_RamGeneralC1_EngineRunningStable_0 := 1409, txt_DbVar_C1_RamGeneralC1_BypassTestCommand_0 := 1410, txt_DbVar_C1_NvOptionsC1_Portillon_0 := 1411, txt_DbVar_C1_NvOptionsC1_Ladder_0 := 1412, txt_DbVar_C1_NvOptionsC1_MeasuringMat_0 := 1413, txt_DbVar_C1_NvOptionsC1_MastDigitalDisplay_0 := 1414, txt_DbVar_C1_NvOptionsC1_Generator_0 := 1415, txt_DbVar_C1_NvOptionsC1_FlashingLightOnRail_0 := 1416, txt_DbVar_C1_NvOptionsC1_AutoStopMeasuringMast_0 := 1417, txt_DbVar_C1_NvOptionsC1_LynxOnAllMvts_0 := 1418, txt_DbVar_C1_NvOptionsC1_WhiteLight15746_0 := 1419, txt_DbVar_C1_NvOptionsC1_AutorisationWorkKeyPresent_0 := 1420, txt_DbVar_C1_NvOptionsC1_FlasingLightAlwaysOnAUS_0 := 1421, txt_DbVar_C1_NvOptionsC1_ContactMastSNCFOption_0 := 1422, txt_DbVar_C1_NvOptionsC1_PresenceContactMast_0 := 1423, txt_DbVar_C1_NvMemoryC1_NvMemoryC_0 := 1424, txt_DbVar_C1_NvMemoryC1_VarMemory1_0 := 1425, txt_DbVar_C1_NvMemoryC1_VarMemory2_0 := 1426, txt_DbVar_C1_NvMemoryC1_VarMemory3_0 := 1427, txt_DbVar_C1_NvMemoryC1_VarMemory4_0 := 1428, txt_DbVar_C1_NvMemoryC1_VarMemory5_0 := 1429, txt_DbVar_C1_NvMemoryC1_VarMemory6_0 := 1430, txt_DbVar_C1_NvMemoryC1_VarMemory7_0 := 1431, txt_DbVar_C1_NvMemoryC1_VarMemory8_0 := 1432, txt_DbVar_C1_NvMemoryC1_VarMemory9_0 := 1433, txt_DbVar_C1_NvMemoryC1_VarMemory10_0 := 1434, txt_DbVar_C1_NvMemoryC1_VarMemory11_0 := 1435, txt_DbVar_C1_NvMemoryC1_VarMemory12_0 := 1436, txt_DbVar_C1_NvMemoryC1_VarMemory13_0 := 1437, txt_DbVar_C1_NvMemoryC1_VarMemory14_0 := 1438, txt_DbVar_C1_NvMemoryC1_CptNbrRegenFinish_0 := 1439, txt_DbVar_C1_NvMemoryC1_FirstKeyNoReloadWithGenerator_0 := 1440, txt_DbVar_C1_NvMemoryC1_NewSocUperReloadWithGenerator_0 := 1441, txt_DbVar_C1_NvMemoryC1_TotalRegenMinutes_0 := 1442, txt_DbVar_C1_NvMemoryC1_TotalElecticMinutes_0 := 1443, txt_DbVar_C1_NvParametersC1_PvgUpDeltaArmTurretPostCmdPrct_0 := 1444, txt_DbVar_C1_NvParametersC1_PvgDownDeltaArmTurretPostCmdPrct_0 := 1445, txt_DbVar_C1_NvParametersC1_PvgUpArrowArmTurretPostCmdPrct_0 := 1446, txt_DbVar_C1_NvParametersC1_PvgDownArrowArmTurretPostCmdPrct_0 := 1447, txt_DbVar_C1_NvParametersC1_PvgInTelescTurretPostCmdPrct_0 := 1448, txt_DbVar_C1_NvParametersC1_PvgOutTelescTurretPostCmdPrct_0 := 1449, txt_DbVar_C1_NvParametersC1_MaxPvgUpDeltaArmCmdPrct_0 := 1450, txt_DbVar_C1_NvParametersC1_MaxPvgDownDeltaArmCmdPrct_0 := 1451, txt_DbVar_C1_NvParametersC1_MaxPvgUpArrowArmCmdPrct_0 := 1452, txt_DbVar_C1_NvParametersC1_MaxPvgDownArrowArmCmdPrct_0 := 1453, txt_DbVar_C1_NvParametersC1_MaxPvgInTelescopeArmCmdPrct_0 := 1454, txt_DbVar_C1_NvParametersC1_MaxPvgOutTelescopeArmCmdPrct_0 := 1455, txt_DbVar_C1_NvParametersC1_MinPvgUpDeltaArmCmdPrct_0 := 1456, txt_DbVar_C1_NvParametersC1_MinPvgDownDeltaArmCmdPrct_0 := 1457, txt_DbVar_C1_NvParametersC1_MinPvgUpArrowArmCmdPrct_0 := 1458, txt_DbVar_C1_NvParametersC1_MinPvgDownArrowArmCmdPrct_0 := 1459, txt_DbVar_C1_NvParametersC1_MinPvgInTelescopeArmCmdPrct_0 := 1460, txt_DbVar_C1_NvParametersC1_MinPvgOutTelescopeArmCmdPrct_0 := 1461, txt_DbVar_C1_NvParametersC1_TresholdAnaToBoForInputs48Xs_0 := 1462, txt_DbVar_C1_NvParametersC1_PvgAxleMovementCmdPrct_0 := 1463, txt_DbVar_C1_NvParametersC1_DeadZoneJoystickTurret_0 := 1464, txt_DbVar_C1_NvParametersC1_DeadZoneJoystickDeltaArm_0 := 1465, txt_DbVar_C1_NvParametersC1_DeadZoneJoystickTelescope_0 := 1466, txt_DbVar_C1_NvParametersC1_DeadZoneJoystickArrow_0 := 1467, txt_DbVar_C1_NvParametersC1_DeadZoneJoystickRailAdvancement_0 := 1468, txt_DbVar_C1_NvParametersC1_DeadZoneJoystickRotationTurret_0 := 1469, txt_DbVar_C1_NvParametersC1_EngineOffCurEvPropMotorAccel_0 := 1470, txt_DbVar_C1_NvParametersC1_MinCurEvPropMotorAccelerator_0 := 1471, txt_DbVar_C1_NvParametersC1_StopCurEvPropMotorAccelerator_0 := 1472, txt_DbVar_C1_NvParametersC1_EngineOffCurEvPropGenerator_0 := 1473, txt_DbVar_C1_NvParametersC1_MinCurEvPropGenerator_0 := 1474, txt_DbVar_C1_NvParametersC1_StopCurEvPropGenerator_0 := 1475, txt_DbVar_C1_NvParametersC1_PidGpEvPropMotorAcc_0 := 1476, txt_DbVar_C1_NvParametersC1_PidTiEvPropMotorAcc_0 := 1477, txt_DbVar_C1_NvParametersC1_PidTdEvPropMotorAcc_0 := 1478, txt_DbVar_C1_NvParametersC1_PidGpEvPropGenerator_0 := 1479, txt_DbVar_C1_NvParametersC1_PidTiEvPropGenerator_0 := 1480, txt_DbVar_C1_NvParametersC1_PidTdEvPropGenerator_0 := 1481, txt_DbVar_C1_NvParametersC1_DeviationLimitTransmPressure_0 := 1482, txt_DbVar_C1_NvParametersC1_OutCharPosDeltaArmAngular_0 := 1483, txt_DbVar_C1_NvParametersC1_OutCharNeuDeltaArmAngular_0 := 1484, txt_DbVar_C1_NvParametersC1_OutCharNegDeltaArmAngular_0 := 1485, txt_DbVar_C1_NvParametersC1_DeviationLimitDeltaArmAngle_0 := 1486, txt_DbVar_C1_NvParametersC1_OutCharPosArrowArmAngular_0 := 1487, txt_DbVar_C1_NvParametersC1_OutCharNeuArrowArmAngular_0 := 1488, txt_DbVar_C1_NvParametersC1_OutCharNegArrowArmAngular_0 := 1489, txt_DbVar_C1_NvParametersC1_DeviationLimitArrowArmAngle_0 := 1490, txt_DbVar_C1_NvParametersC1_MinPvgUpPendularTurretPost_0 := 1491, txt_DbVar_C1_NvParametersC1_MinPvgUpPendularNacellePost_0 := 1492, txt_DbVar_C1_NvParametersC1_MinPvgUpPendularRadioPost_0 := 1493, txt_DbVar_C1_NvParametersC1_MaxPvgUpPendularTurretPost_0 := 1494, txt_DbVar_C1_NvParametersC1_MaxPvgUpPendularNacellePost_0 := 1495, txt_DbVar_C1_NvParametersC1_MaxPvgUpPendularRadioPost_0 := 1496, txt_DbVarArrDescr_C1_NvParametersC1_UpPendularRampRatioTurret := 1497, txt_DbVar_C1_NvParametersC1_UpPendularRampRatioTurret_0 := 1498, txt_DbVar_C1_NvParametersC1_UpPendularRampRatioTurret_1 := 1499, txt_DbVarArrDescr_C1_NvParametersC1_UpPendularRampRatioNacelle := 1500, txt_DbVar_C1_NvParametersC1_UpPendularRampRatioNacelle_0 := 1501, txt_DbVar_C1_NvParametersC1_UpPendularRampRatioNacelle_1 := 1502, txt_DbVarArrDescr_C1_NvParametersC1_UpPendularRampRatioRadio := 1503, txt_DbVar_C1_NvParametersC1_UpPendularRampRatioRadio_0 := 1504, txt_DbVar_C1_NvParametersC1_UpPendularRampRatioRadio_1 := 1505, txt_DbVar_C1_NvParametersC1_MinPvgDownPendularTurretPost_0 := 1506, txt_DbVar_C1_NvParametersC1_MinPvgDownPendularNacellePost_0 := 1507, txt_DbVar_C1_NvParametersC1_MinPvgDownPendularRadioPost_0 := 1508, txt_DbVar_C1_NvParametersC1_MaxPvgDownPendularTurretPost_0 := 1509, txt_DbVar_C1_NvParametersC1_MaxPvgDownPendularNacellePost_0 := 1510, txt_DbVar_C1_NvParametersC1_MaxPvgDownPendularRadioPost_0 := 1511, txt_DbVarArrDescr_C1_NvParametersC1_DownPendularRampRatioTurret := 1512, txt_DbVar_C1_NvParametersC1_DownPendularRampRatioTurret_0 := 1513, txt_DbVar_C1_NvParametersC1_DownPendularRampRatioTurret_1 := 1514, txt_DbVarArrDescr_C1_NvParametersC1_DownPendularRampRatioNacelle := 1515, txt_DbVar_C1_NvParametersC1_DownPendularRampRatioNacelle_0 := 1516, txt_DbVar_C1_NvParametersC1_DownPendularRampRatioNacelle_1 := 1517, txt_DbVarArrDescr_C1_NvParametersC1_DownPendularRampRatioRadio := 1518, txt_DbVar_C1_NvParametersC1_DownPendularRampRatioRadio_0 := 1519, txt_DbVar_C1_NvParametersC1_DownPendularRampRatioRadio_1 := 1520, txt_DbVar_C1_NvParametersC1_MinPvgUpIncliBasketTurretPost_0 := 1521, txt_DbVar_C1_NvParametersC1_MinPvgUpIncliBasketNacellePost_0 := 1522, txt_DbVar_C1_NvParametersC1_MinPvgUpIncliBasketRadioPost_0 := 1523, txt_DbVar_C1_NvParametersC1_MaxPvgUpIncliBasketTurretPost_0 := 1524, txt_DbVar_C1_NvParametersC1_MaxPvgUpIncliBasketNacellePost_0 := 1525, txt_DbVar_C1_NvParametersC1_MaxPvgUpIncliBasketRadioPost_0 := 1526, txt_DbVarArrDescr_C1_NvParametersC1_UpInclinBasketRampRatioTurret := 1527, txt_DbVar_C1_NvParametersC1_UpInclinBasketRampRatioTurret_0 := 1528, txt_DbVar_C1_NvParametersC1_UpInclinBasketRampRatioTurret_1 := 1529, txt_DbVarArrDescr_C1_NvParametersC1_UpInclinBasketRampRatioNacelle := 1530, txt_DbVar_C1_NvParametersC1_UpInclinBasketRampRatioNacelle_0 := 1531, txt_DbVar_C1_NvParametersC1_UpInclinBasketRampRatioNacelle_1 := 1532, txt_DbVarArrDescr_C1_NvParametersC1_UpInclinBasketRampRatioRadio := 1533, txt_DbVar_C1_NvParametersC1_UpInclinBasketRampRatioRadio_0 := 1534, txt_DbVar_C1_NvParametersC1_UpInclinBasketRampRatioRadio_1 := 1535, txt_DbVar_C1_NvParametersC1_MinPvgDownIncliBasketTurretPost_0 := 1536, txt_DbVar_C1_NvParametersC1_MinPvgDownIncliBasketNacellePost_0 := 1537, txt_DbVar_C1_NvParametersC1_MinPvgDownIncliBasketRadioPost_0 := 1538, txt_DbVar_C1_NvParametersC1_MaxPvgDownIncliBasketTurretPost_0 := 1539, txt_DbVar_C1_NvParametersC1_MaxPvgDownIncliBasketNacellePost_0 := 1540, txt_DbVar_C1_NvParametersC1_MaxPvgDownIncliBasketRadioPost_0 := 1541, txt_DbVarArrDescr_C1_NvParametersC1_DownInclinBasketRampRatioTurret := 1542, txt_DbVar_C1_NvParametersC1_DownInclinBasketRampRatioTurret_0 := 1543, txt_DbVar_C1_NvParametersC1_DownInclinBasketRampRatioTurret_1 := 1544, txt_DbVarArrDescr_C1_NvParametersC1_DownInclinBasketRampRatioNacelle := 1545, txt_DbVar_C1_NvParametersC1_DownInclinBasketRampRatioNacelle_0 := 1546, txt_DbVar_C1_NvParametersC1_DownInclinBasketRampRatioNacelle_1 := 1547, txt_DbVarArrDescr_C1_NvParametersC1_DownInclinBasketRampRatioRadio := 1548, txt_DbVar_C1_NvParametersC1_DownInclinBasketRampRatioRadio_0 := 1549, txt_DbVar_C1_NvParametersC1_DownInclinBasketRampRatioRadio_1 := 1550, txt_DbVar_C1_NvParametersC1_MinPvgRotBasktClkwiseTurretPost_0 := 1551, txt_DbVar_C1_NvParametersC1_MinPvgRotBasktClkwiseNacellePost_0 := 1552, txt_DbVar_C1_NvParametersC1_MinPvgRotBasketClkwiseRadioPost_0 := 1553, txt_DbVar_C1_NvParametersC1_MaxPvgRotBasketClkwiseTurretPost_0 := 1554, txt_DbVar_C1_NvParametersC1_MaxPvgRotBasktClkwiseNacellePost_0 := 1555, txt_DbVar_C1_NvParametersC1_MaxPvgRotBasketClkwiseRadioPost_0 := 1556, txt_DbVarArrDescr_C1_NvParametersC1_RotBasketClkwiseRampRatioTurret := 1557, txt_DbVar_C1_NvParametersC1_RotBasketClkwiseRampRatioTurret_0 := 1558, txt_DbVar_C1_NvParametersC1_RotBasketClkwiseRampRatioTurret_1 := 1559, txt_DbVarArrDescr_C1_NvParametersC1_RotBasketClkwiseRampRatioNacel := 1560, txt_DbVar_C1_NvParametersC1_RotBasketClkwiseRampRatioNacel_0 := 1561, txt_DbVar_C1_NvParametersC1_RotBasketClkwiseRampRatioNacel_1 := 1562, txt_DbVarArrDescr_C1_NvParametersC1_RotBasketClkwiseRampRatioRadio := 1563, txt_DbVar_C1_NvParametersC1_RotBasketClkwiseRampRatioRadio_0 := 1564, txt_DbVar_C1_NvParametersC1_RotBasketClkwiseRampRatioRadio_1 := 1565, txt_DbVar_C1_NvParametersC1_MinPvgRotBasktCtClkwiseTurtPost_0 := 1566, txt_DbVar_C1_NvParametersC1_MinPvgRotBasktCtClkwiseNacelPost_0 := 1567, txt_DbVar_C1_NvParametersC1_MinPvgRotBasktCtClkwiseRadioPost_0 := 1568, txt_DbVar_C1_NvParametersC1_MaxPvgRotBasktCtClkwiseTuretPost_0 := 1569, txt_DbVar_C1_NvParametersC1_MaxPvgRotBasktCtClkwiseNacelPost_0 := 1570, txt_DbVar_C1_NvParametersC1_MaxPvgRotBasktCtClkwiseRadioPost_0 := 1571, txt_DbVarArrDescr_C1_NvParametersC1_RotBasketCtClkwiseRampRatioTuret := 1572, txt_DbVar_C1_NvParametersC1_RotBasketCtClkwiseRampRatioTuret_0 := 1573, txt_DbVar_C1_NvParametersC1_RotBasketCtClkwiseRampRatioTuret_1 := 1574, txt_DbVarArrDescr_C1_NvParametersC1_RotBasketCtClkwiseRampRatioNacel := 1575, txt_DbVar_C1_NvParametersC1_RotBasketCtClkwiseRampRatioNacel_0 := 1576, txt_DbVar_C1_NvParametersC1_RotBasketCtClkwiseRampRatioNacel_1 := 1577, txt_DbVarArrDescr_C1_NvParametersC1_RotBasketCtClkwiseRampRatioRadio := 1578, txt_DbVar_C1_NvParametersC1_RotBasketCtClkwiseRampRatioRadio_0 := 1579, txt_DbVar_C1_NvParametersC1_RotBasketCtClkwiseRampRatioRadio_1 := 1580, txt_DbVar_C1_NvParametersC1_MinPvgRotTurretClkwiseTurretPost_0 := 1581, txt_DbVar_C1_NvParametersC1_MinPvgRotTurretClkwiseNacelPost_0 := 1582, txt_DbVar_C1_NvParametersC1_MinPvgRotTurretClkwiseRadioPost_0 := 1583, txt_DbVar_C1_NvParametersC1_MaxPvgRotTurretClkwiseTurretPost_0 := 1584, txt_DbVar_C1_NvParametersC1_MaxPvgRotTurretClkwiseNacelPost_0 := 1585, txt_DbVar_C1_NvParametersC1_MaxPvgRotTurretClkwiseRadioPost_0 := 1586, txt_DbVarArrDescr_C1_NvParametersC1_RotTurretClkwiseRampRatioTurret := 1587, txt_DbVar_C1_NvParametersC1_RotTurretClkwiseRampRatioTurret_0 := 1588, txt_DbVar_C1_NvParametersC1_RotTurretClkwiseRampRatioTurret_1 := 1589, txt_DbVarArrDescr_C1_NvParametersC1_RotTurretClkwiseRampRatioNacelle := 1590, txt_DbVar_C1_NvParametersC1_RotTurretClkwiseRampRatioNacelle_0 := 1591, txt_DbVar_C1_NvParametersC1_RotTurretClkwiseRampRatioNacelle_1 := 1592, txt_DbVarArrDescr_C1_NvParametersC1_RotTurretClkwiseRampRatioRadio := 1593, txt_DbVar_C1_NvParametersC1_RotTurretClkwiseRampRatioRadio_0 := 1594, txt_DbVar_C1_NvParametersC1_RotTurretClkwiseRampRatioRadio_1 := 1595, txt_DbVar_C1_NvParametersC1_MinPvgRotTurretCtClkwiseTurtPost_0 := 1596, txt_DbVar_C1_NvParametersC1_MinPvgRotTurretCtClkwseNacelPost_0 := 1597, txt_DbVar_C1_NvParametersC1_MinPvgRotTuretCtClkwseRadioPost_0 := 1598, txt_DbVar_C1_NvParametersC1_MaxPvgRotTurretCtClkwseTuretPost_0 := 1599, txt_DbVar_C1_NvParametersC1_MaxPvgRotTurretCtClkwseNacelPost_0 := 